(* CODESYS project LABELIX_849_HSC_Rtrig_24juillet.project
   CustomField04_name: CustomField04
   CustomField06_name: CustomField06
   CustomField07_name: CustomField07
   CustomField09_name: CustomField09
   CustomField08_name: CustomField08
   CustomField02_name: CustomField02
   CustomField05_name: CustomField05
   CustomField01_name: CustomField01
   CustomField03_name: CustomField03
   CustomField10_name: CustomField10

Project tree, tasks and I/O mapping:
  HMIS5T_REWIND : HMIS5T, Schneider Electric, order no. HMIS5T, version 2.0.3.24
    HMI Application
    COM1
      SoMachine_Network_Manager1 : SoMachine-Network_Manager, Schneider Electric, version 2.0.0.1
    USB
      SoMachine_Network_Manager3 : SoMachine-Network_Manager, Schneider Electric, version 2.0.0.1
    Ethernet
      SoMachine_Network_Manager2 : SoMachine-Network_Manager, Schneider Electric, version 2.0.0.1
  HMIS5T : HMIS5T, Schneider Electric, order no. HMIS5T, version 2.0.3.24
    HMI Application
    COM1
      SoMachine_Network_Manager4 : SoMachine-Network_Manager, Schneider Electric, version 2.0.0.1
    USB
      SoMachine_Network_Manager6 : SoMachine-Network_Manager, Schneider Electric, version 2.0.0.1
    Ethernet
      SoMachine_Network_Manager5 : SoMachine-Network_Manager, Schneider Electric, version 2.0.0.1
  MyController : TM258LF42DR, Schneider Electric, order no. TM258LF42DR, version 2.0.31.14
    application Application
      libraries: Toolbox, 2.0.3.1 (Schneider Electric)
      task MAST (cyclic, interval t#10ms, priority 2) calls PLC_PRG_LD_1
      task TaskMain (cyclic, interval t#20ms, priority 3) calls AccessCode, CAN_NETWORK, CONVERT, DRYER_1FD_3FX_STATIONS, ETH_NETWORK, FAULT_INTERLOCK, GRAVURE_PGM, LATCH_ERROR, Main, UNWIND_TENS_CTRL, COUNTER, UNWIND_TENS_CTRL, UW_FILT, UW_DIAM
      task Event_Task (externalevent, external event BLOCK0_I0, priority 1) calls EVENT_TASK
      COUNTER/
        program SPEED_DISPLAY [CFC]
        program PLC_PRG_LD_1 [LD]
        program speed_task [ST]
        program COUNTER [ST]
        program PLC_PRG_LD [LD]
      global variables GVL_OLD
      program Main [LD]
      global variables GVL_ARCHIVE
      global variables GVL_CAN_ARRAY
      program ETH_NETWORK [ST]
      global variables GVL_GENERAL
      program FAULT_INTERLOCK [LD]
      global variables GVL_ENCODER
      global variables GVL_NOT_USED_IOs
      global variables GVL_HMI
      program EVENT_TASK [ST]
      Symbols
      function HiddenPOU [ST]
      global variables GVL_ETHERNET
      data type stDryingGroup
      ErrorProvider
      program CONVERT [ST]
      program DRYER_1FD_3FX_STATIONS [LD]
      program CAN_NETWORK [ST]
      global variables GVL_KEEP_ARRAY
      program GRAVURE_PGM [LD]
      data type stTensionCtrlState
      global variables GVL_CONVERT
      data type stFlexoStation
      global variables GVL_KEY
      global variables GVL_DEBUG
      program LATCH_ERROR [LD]
      OPTIONS/
        program AccessCode [ST]
      UNWIND/
        program UW_FILT [LD]
        program UNWIND_TENS_CTRL [CFC]
        program UW_DIAM [ST]
      global variables GVL_counter
    Ethernet
        settings: IPAddress = [192, 168, 100, 202]; SubnetMask = [255, 255, 255, 0]; GatewayAddress = [192, 168, 100, 254]; WebServer = TRUE
      Modbus_TCP_Master : Modbus TCP Master, 3S - Smart Software Solutions GmbH, version 3.4.1.0
        GRAVURE : Modbus TCP Slave, 3S - Smart Software Solutions GmbH, version 3.4.0.0
            settings: IPAddress = [192, 168, 100, 208]; GravureWrite.Function Code = 16; GravureWrite.Read Offset = 0; GravureWrite.Read Length = 0; GravureWrite.Write Offset = 16#072C; GravureWrite.Write Length = 4; GravureWrite.Cycle Time = 100
            output wPar1837_GravureOn_ETH : WORD  // GravureWrite
            output wPar1838_GravureProcessOn_ETH : WORD  // GravureWrite
            output wPar1839_GravureFWD_ETH : WORD  // GravureWrite
            output wPar1840_GravureBCK_ETH : WORD  // GravureWrite
        REWIND_DF : Modbus TCP Slave, 3S - Smart Software Solutions GmbH, version 3.4.0.0
            settings: IPAddress = [192, 168, 100, 210]; REWIND_READ.Function Code = 3; REWIND_READ.Read Offset = 16#07E2; REWIND_READ.Read Length = 1; REWIND_READ.Write Offset = 0; REWIND_READ.Write Length = 0; REWIND_READ.Cycle Time = 100; RewindON.Function Code = 16; RewindON.Read Offset = 0; RewindON.Read Length = 0; RewindON.Write Offset = 16#072C; RewindON.Write Length = 2; RewindON.Cycle Time = 100; REWIND_STATE.Function Code = 3; REWIND_STATE.Read Offset = 16#03E8; REWIND_STATE.Read Length = 3; REWIND_STATE.Write Offset = 0; REWIND_STATE.Write Length = 0; REWIND_STATE.Cycle Time = 100
            input  wPar2019_DryPermit_ETH : WORD  // REWIND_READ
            output wPar1837_RewindOn_ETH : WORD  // RewindON
            output wPar1838_PidOn_ETH : WORD  // RewindON
            input  wPar1001_RewindHealthy_ETH : WORD  // REWIND_STATE
            input  wPar1002_RewindActive_ETH : WORD  // REWIND_STATE
            input  wPar1003_RewindZeroSpd_ETH : WORD  // REWIND_STATE
        REWIND : Modbus TCP Slave, 3S - Smart Software Solutions GmbH, version 3.4.0.0
            settings: IPAddress = [192, 168, 100, 204]; REWIND_READ.Function Code = 3; REWIND_READ.Read Offset = 16#07E2; REWIND_READ.Read Length = 1; REWIND_READ.Write Offset = 0; REWIND_READ.Write Length = 0; REWIND_READ.Cycle Time = 100; RewindON.Function Code = 16; RewindON.Read Offset = 0; RewindON.Read Length = 0; RewindON.Write Offset = 16#072C; RewindON.Write Length = 2; RewindON.Cycle Time = 100; REWIND_STATE.Function Code = 3; REWIND_STATE.Read Offset = 16#03E8; REWIND_STATE.Read Length = 3; REWIND_STATE.Write Offset = 0; REWIND_STATE.Write Length = 0; REWIND_STATE.Cycle Time = 100
            input  wPar2019_DryPermit_ETH : WORD  // REWIND_READ
            output wPar1837_RewindOn_ETH : WORD  // RewindON
            output wPar1838_PidOn_ETH : WORD  // RewindON
            input  wPar1001_RewindHealthy_ETH : WORD  // REWIND_STATE
            input  wPar1002_RewindActive_ETH : WORD  // REWIND_STATE
            input  wPar1003_RewindZeroSpd_ETH : WORD  // REWIND_STATE
        INFEED : Modbus TCP Slave, 3S - Smart Software Solutions GmbH, version 3.4.0.0
            settings: IPAddress = [192, 168, 100, 203]; Channel 2.Function Code = 16; Channel 2.Read Offset = 0; Channel 2.Read Length = 0; Channel 2.Write Offset = 16#072C; Channel 2.Write Length = 2; Channel 2.Cycle Time = 100; ALL_UnidriveSPs.Function Code = 3; ALL_UnidriveSPs.Read Offset = 16#07EF; ALL_UnidriveSPs.Read Length = 1; ALL_UnidriveSPs.Write Offset = 0; ALL_UnidriveSPs.Write Length = 0; ALL_UnidriveSPs.Cycle Time = 100; INFEED_STATE.Function Code = 3; INFEED_STATE.Read Offset = 16#03E8; INFEED_STATE.Read Length = 3; INFEED_STATE.Write Offset = 0; INFEED_STATE.Write Length = 0; INFEED_STATE.Cycle Time = 100; CounterReached_ETH.Function Code = 3; CounterReached_ETH.Read Offset = 16#078C; CounterReached_ETH.Read Length = 1; CounterReached_ETH.Write Offset = 0; CounterReached_ETH.Write Length = 0; CounterReached_ETH.Cycle Time = 100
            output wPar1837_InfeedOn_ETH : WORD  // Channel 2
            output wPar1838_FilterOn_ETH : WORD  // Channel 2
            input  wReadReg2031 : WORD  // ALL_UnidriveSPs
            input  wPar1001_InfeedHealthy_ETH : WORD  // INFEED_STATE
            input  wPar1002_InfeedActive_ETH : WORD  // INFEED_STATE
            input  wPar1003_InfeedZeroSpd_ETH : WORD  // INFEED_STATE
            input  wPar1933_CountReach_ETH : WORD  // CounterReached_ETH
        ANILOX_2 : Modbus TCP Slave, 3S - Smart Software Solutions GmbH, version 3.4.0.0
            settings: IPAddress = [192, 168, 100, 207]; AniloxWrite.Function Code = 16; AniloxWrite.Read Offset = 0; AniloxWrite.Read Length = 0; AniloxWrite.Write Offset = 16#072C; AniloxWrite.Write Length = 4; AniloxWrite.Cycle Time = 100
            output wPar1837_AniloxOn_2_ETH : WORD  // AniloxWrite
            output wPar1838_ProcessOn_2_ETH : WORD  // AniloxWrite
            output wPar1839_AniloxFWD_2_ETH : WORD  // AniloxWrite
            output wPar1840_AniloxBCK_2_ETH : WORD  // AniloxWrite
        TOP_REWIND : Modbus TCP Slave, 3S - Smart Software Solutions GmbH, version 3.4.0.0
            settings: IPAddress = [192, 168, 100, 205]; TOP_REWIND_READ.Function Code = 3; TOP_REWIND_READ.Read Offset = 16#07E2; TOP_REWIND_READ.Read Length = 1; TOP_REWIND_READ.Write Offset = 0; TOP_REWIND_READ.Write Length = 0; TOP_REWIND_READ.Cycle Time = 100; TopRewindON.Function Code = 16; TopRewindON.Read Offset = 0; TopRewindON.Read Length = 0; TopRewindON.Write Offset = 16#072C; TopRewindON.Write Length = 2; TopRewindON.Cycle Time = 100; TOP_REWIND_STATE.Function Code = 3; TOP_REWIND_STATE.Read Offset = 16#03E8; TOP_REWIND_STATE.Read Length = 3; TOP_REWIND_STATE.Write Offset = 0; TOP_REWIND_STATE.Write Length = 0; TOP_REWIND_STATE.Cycle Time = 100
            input  wPar2019 : WORD  // TOP_REWIND_READ
            output wPar1837_TopRewindOn_ETH : WORD  // TopRewindON
            output wPar1838_TopPidOn_ETH : WORD  // TopRewindON
            input  wPar1001_TopRewindHealthy_ETH : WORD  // TOP_REWIND_STATE
            input  wPar1002_TopRewindActive_ETH : WORD  // TOP_REWIND_STATE
            input  wPar1003_TopRewindZeroSpd_ETH : WORD  // TOP_REWIND_STATE
        REXROTH_1 : Modbus TCP Slave, 3S - Smart Software Solutions GmbH, version 3.4.0.0
            settings: IPAddress = [192, 168, 100, 211]; Channel 1.Function Code = 3; Channel 1.Read Offset = 16#0000; Channel 1.Read Length = 10; Channel 1.Write Offset = 0; Channel 1.Write Length = 0; Channel 1.Cycle Time = 100; Channel 2.Function Code = 16; Channel 2.Read Offset = 0; Channel 2.Read Length = 0; Channel 2.Write Offset = 16#000A; Channel 2.Write Length = 10; Channel 2.Cycle Time = 100
            output bGravureComTriggerRead : BIT  // Channel 1
            input  wInfeedManualGearing_ETH_i : WORD  // Channel 1
            input  wGravureGearingAdjust : WORD  // Channel 1
            input  bGravure_StatusDisabled_HMI_q2 : BOOL  // Channel 1.Bit 0
            input  bGravure_StatusSlowRot_HMI_q2 : BOOL  // Channel 1.Bit 1
            input  bGravure_StatusSynch_HMI_q2 : BOOL  // Channel 1.Bit 2
            input  bGravure_StatusError_HMI_q2 : BOOL  // Channel 1.Bit 3
            input  wDeviation_low_gb : WORD  // Channel 1
            input  wDeviation_high_gb : WORD  // Channel 1
            input  wRegiCtrlSetpoint_low_gb : WORD  // Channel 1
            input  wRegiCtrlSetpoint_high_gb : WORD  // Channel 1
            input  wLoadcellTension_low_gb : WORD  // Channel 1
            input  wLoadcellTension_high_gb : WORD  // Channel 1
            input  bInfeed_StatusDisabled_ETH_q : BOOL  // Channel 1.Bit 0
            input  bInfeed_StatusSlowRot_ETH_q : BOOL  // Channel 1.Bit 1
            input  bInfeed_StatusSynch_ETH_q : BOOL  // Channel 1.Bit 2
            input  bInfeed_StatusError_ETH_q : BOOL  // Channel 1.Bit 3
            output bGravureComTriggerWrite : BIT  // Channel 2
            output bGravure_Tens_Inc_ETH_q : BOOL  // Channel 2.Bit 0
            output bGravure_Tens_Dec_ETH_q : BOOL  // Channel 2.Bit 1
            output bGravure_Reg_Adv_ETH_q : BOOL  // Channel 2.Bit 2
            output bGravure_Reg_Ret_ETH_q : BOOL  // Channel 2.Bit 3
            output bGravureOn_ETH_q : BOOL  // Channel 2.Bit 4
            output bGravure_ResetDrive_HMI_q : BOOL  // Channel 2.Bit 5
            output bRewindPID_Out : BOOL  // Channel 2.Bit 6
            output bGravureSlowRot_ETH_q : BOOL  // Channel 2.Bit 7
            output bGravureRegiOn_HMI_q : BOOL  // Channel 2.Bit 8
            output bGravure_Jog_Adv_HMI_q : BOOL  // Channel 2.Bit 9
            output bGravure_Jog_Ret_HMI_q : BOOL  // Channel 2.Bit 10
            output bInfeedRegiOn_HMI_q : BOOL  // Channel 2.Bit 11
            output bInfeed_Tens_Inc_ETH_i : BOOL  // Channel 2.Bit 0
            output bInfeed_Tens_dec_ETH_i : BOOL  // Channel 2.Bit 1
            output bInfeedOn_ETH_i : BOOL  // Channel 2.Bit 2
            output bInfeed_Manual_ETH_i : BOOL  // Channel 2.Bit 3
            output bInfeed_ResetDrive_ETH_i : BOOL  // Channel 2.Bit 4
            output wRegAdjustStep_low_gb : WORD  // Channel 2
            output wRegAdjustStep_high_gb : WORD  // Channel 2
            unmapped channels: Channel 1, Channel 1, Channel 2, Channel 2, Channel 2, Channel 2, Channel 2, Channel 2, Channel 2, Channel 2
        ANILOX_1 : Modbus TCP Slave, 3S - Smart Software Solutions GmbH, version 3.4.0.0
            settings: IPAddress = [192, 168, 100, 206]; AniloxWrite.Function Code = 16; AniloxWrite.Read Offset = 0; AniloxWrite.Read Length = 0; AniloxWrite.Write Offset = 16#072C; AniloxWrite.Write Length = 4; AniloxWrite.Cycle Time = 100
            output wPar1837_AniloxOn_ETH : WORD  // AniloxWrite
            output wPar1838_ProcessOn_ETH : WORD  // AniloxWrite
            output wPar1839_AniloxFWD_ETH : WORD  // AniloxWrite
            output wPar1840_AniloxBCK_ETH : WORD  // AniloxWrite
    CAN0
      CANopen_Performance : CANopen Performance, Schneider Electric, order no. 1806, version 3.0.0.9
          settings: Enable Sync generation = FALSE; Enable Heartbeat generation = FALSE
        STATION_BOARD1 : OTB 1C0DM9LP, Schneider Electric, order no. 65275, version ProductVersion=0, ProductRevision=65537, Filename=SEOTB1C0DM9LP_0100E, FileVersion=1, FileRevision=0
            settings: General Options.Optional Device = TRUE; General Options.Not initialize = TRUE; NODEIDSAVED = 21; SDO Timeout = 1000000; EXPERTSETTINGS = True; Emergency-General Parameters.Emergency enabled = FALSE; Emergency-General Parameters.Emergency COBID = 16#95; Heartbeat-Producer Time = 200; PDO 16#1400.COBID = 16#00000215; PDO 16#1401.COBID = 16#80000315; PDO 16#1402.COBID = 16#80000415; PDO 16#1403.COBID = 16#80000515; PDO 16#1800.COBID = 16#00000195; PDO 16#1801.COBID = 16#80000295; PDO 16#1802.COBID = 16#80000395; PDO 16#1803.COBID = 16#80000495; Word Write Output 0 to 7.Index = 16#6300; Word Write Output 0 to 7.Subindex = 16#01; Word Write Output 0 to 7.ObjectLength = 16; Word Read Input 0 to 11.Index = 16#6100; Word Read Input 0 to 11.Subindex = 16#01; Word Read Input 0 to 11.ObjectLength = 16; Number of SDO = 33; Set Guardtime.Index = 16#100C; Set Guardtime.Subindex = 16#00; Set Guardtime.Value = 16#00000000; Set Guardtime.Size = 16; Set Guardtime.AbortIfError = FALSE; Set Guardtime.JumpToLine = FALSE; Set Guardtime.Line = 0; Set Lifetime.Index = 16#100D; Set Lifetime.Subindex = 16#00; Set Lifetime.Value = 16#00000000; Set Lifetime.Size = 8; Set Lifetime.AbortIfError = FALSE; Set Lifetime.JumpToLine = FALSE; Set Lifetime.Line = 0; Set Emcy CobID.Index = 16#1014; Set Emcy CobID.Subindex = 16#00; Set Emcy CobID.Value = 16#80000095;
              Set Emcy CobID.Size = 32; Set Emcy CobID.AbortIfError = FALSE; Set Emcy CobID.JumpToLine = FALSE; Set Emcy CobID.Line = 0; Set Heartbeat Consumer.Index = 16#1016; Set Heartbeat Consumer.Subindex = 16#01; Set Heartbeat Consumer.Value = 0; Set Heartbeat Consumer.Size = 32; Set Heartbeat Consumer.AbortIfError = FALSE; Set Heartbeat Consumer.JumpToLine = FALSE; Set Heartbeat Consumer.Line = 0; Set Heartbeat Producer.Index = 16#1017; Set Heartbeat Producer.Subindex = 16#00; Set Heartbeat Producer.Value = 16#000000C8; Set Heartbeat Producer.Size = 16; Set Heartbeat Producer.AbortIfError = FALSE; Set Heartbeat Producer.JumpToLine = FALSE; Set Heartbeat Producer.Line = 0; Disable PDO.Index = 16#1400; Disable PDO.Subindex = 16#01; Disable PDO.Value = 16#80000215; Disable PDO.Size = 32; Disable PDO.AbortIfError = FALSE; Disable PDO.JumpToLine = FALSE; Disable PDO.Line = 0; Set transmission type.Index = 16#1400; Set transmission type.Subindex = 16#02; Set transmission type.Value = 16#FF; Set transmission type.Size = 8; Set transmission type.AbortIfError = FALSE; Set transmission type.JumpToLine = FALSE; Set transmission type.Line = 0; Clear pdo mapping.Index = 16#1600; Clear pdo mapping.Subindex = 16#00; Clear pdo mapping.Value = 16#0; Clear pdo mapping.Size = 8; Clear pdo mapping.AbortIfError = FALSE; Clear pdo mapping.JumpToLine = FALSE; Clear pdo mapping.Line = 0; Set Mapping.Index = 16#1600;
              Set Mapping.Subindex = 16#01; Set Mapping.Value = 16#63000110; Set Mapping.Size = 32; Set Mapping.AbortIfError = FALSE; Set Mapping.JumpToLine = FALSE; Set Mapping.Line = 0; Set number of pdos.Index = 16#1600; Set number of pdos.Subindex = 16#00; Set number of pdos.Value = 16#01; Set number of pdos.Size = 8; Set number of pdos.AbortIfError = FALSE; Set number of pdos.JumpToLine = FALSE; Set number of pdos.Line = 0; Set and enable COB-ID.Index = 16#1400; Set and enable COB-ID.Subindex = 16#01; Set and enable COB-ID.Value = 16#00000215; Set and enable COB-ID.Size = 32; Set and enable COB-ID.AbortIfError = FALSE; Set and enable COB-ID.JumpToLine = FALSE; Set and enable COB-ID.Line = 0; Disable PDO.Index = 16#1401; Disable PDO.Subindex = 16#01; Disable PDO.Value = 16#80000315; Disable PDO.Size = 32; Disable PDO.AbortIfError = FALSE; Disable PDO.JumpToLine = FALSE; Disable PDO.Line = 0; Disable PDO.Index = 16#1402; Disable PDO.Subindex = 16#01; Disable PDO.Value = 16#80000415; Disable PDO.Size = 32; Disable PDO.AbortIfError = FALSE; Disable PDO.JumpToLine = FALSE; Disable PDO.Line = 0; Disable PDO.Index = 16#1403; Disable PDO.Subindex = 16#01; Disable PDO.Value = 16#80000515; Disable PDO.Size = 32; Disable PDO.AbortIfError = FALSE; Disable PDO.JumpToLine = FALSE;
              Disable PDO.Line = 0; Disable PDO.Index = 16#1404; Disable PDO.Subindex = 16#01; Disable PDO.Value = 16#80000001; Disable PDO.Size = 32; Disable PDO.AbortIfError = FALSE; Disable PDO.JumpToLine = FALSE; Disable PDO.Line = 0; Disable PDO.Index = 16#1405; Disable PDO.Subindex = 16#01; Disable PDO.Value = 16#80000001; Disable PDO.Size = 32; Disable PDO.AbortIfError = FALSE; Disable PDO.JumpToLine = FALSE; Disable PDO.Line = 0; Disable PDO.Index = 16#1406; Disable PDO.Subindex = 16#01; Disable PDO.Value = 16#80000001; Disable PDO.Size = 32; Disable PDO.AbortIfError = FALSE; Disable PDO.JumpToLine = FALSE; Disable PDO.Line = 0; Disable PDO.Index = 16#1407; Disable PDO.Subindex = 16#01; Disable PDO.Value = 16#80000001; Disable PDO.Size = 32; Disable PDO.AbortIfError = FALSE; Disable PDO.JumpToLine = FALSE; Disable PDO.Line = 0; Disable PDO.Index = 16#1800; Disable PDO.Subindex = 16#01; Disable PDO.Value = 16#80000195; Disable PDO.Size = 32; Disable PDO.AbortIfError = FALSE; Disable PDO.JumpToLine = FALSE; Disable PDO.Line = 0; Set transmission type.Index = 16#1800; Set transmission type.Subindex = 16#02; Set transmission type.Value = 16#FF; Set transmission type.Size = 8;
              Set transmission type.AbortIfError = FALSE; Set transmission type.JumpToLine = FALSE; Set transmission type.Line = 0; Set inhibit time.Index = 16#1800; Set inhibit time.Subindex = 16#03; Set inhibit time.Value = 16#0000; Set inhibit time.Size = 16; Set inhibit time.AbortIfError = FALSE; Set inhibit time.JumpToLine = FALSE; Set inhibit time.Line = 0; Set event time.Index = 16#1800; Set event time.Subindex = 16#05; Set event time.Value = 16#0000; Set event time.Size = 16; Set event time.AbortIfError = FALSE; Set event time.JumpToLine = FALSE; Set event time.Line = 0; Clear pdo mapping.Index = 16#1A00; Clear pdo mapping.Subindex = 16#00; Clear pdo mapping.Value = 16#0; Clear pdo mapping.Size = 8; Clear pdo mapping.AbortIfError = FALSE; Clear pdo mapping.JumpToLine = FALSE; Clear pdo mapping.Line = 0; Set Mapping.Index = 16#1A00; Set Mapping.Subindex = 16#01; Set Mapping.Value = 16#61000110; Set Mapping.Size = 32; Set Mapping.AbortIfError = FALSE; Set Mapping.JumpToLine = FALSE; Set Mapping.Line = 0; Set number of pdos.Index = 16#1A00; Set number of pdos.Subindex = 16#00; Set number of pdos.Value = 16#01; Set number of pdos.Size = 8; Set number of pdos.AbortIfError = FALSE; Set number of pdos.JumpToLine = FALSE; Set number of pdos.Line = 0; Set and enable COB-ID.Index = 16#1800; Set and enable COB-ID.Subindex = 16#01;
              Set and enable COB-ID.Value = 16#00000195; Set and enable COB-ID.Size = 32; Set and enable COB-ID.AbortIfError = FALSE; Set and enable COB-ID.JumpToLine = FALSE; Set and enable COB-ID.Line = 0; Disable PDO.Index = 16#1801; Disable PDO.Subindex = 16#01; Disable PDO.Value = 16#80000295; Disable PDO.Size = 32; Disable PDO.AbortIfError = FALSE; Disable PDO.JumpToLine = FALSE; Disable PDO.Line = 0; Disable PDO.Index = 16#1802; Disable PDO.Subindex = 16#01; Disable PDO.Value = 16#80000395; Disable PDO.Size = 32; Disable PDO.AbortIfError = FALSE; Disable PDO.JumpToLine = FALSE; Disable PDO.Line = 0; Disable PDO.Index = 16#1803; Disable PDO.Subindex = 16#01; Disable PDO.Value = 16#80000495; Disable PDO.Size = 32; Disable PDO.AbortIfError = FALSE; Disable PDO.JumpToLine = FALSE; Disable PDO.Line = 0; Disable PDO.Index = 16#1804; Disable PDO.Subindex = 16#01; Disable PDO.Value = 16#80000001; Disable PDO.Size = 32; Disable PDO.AbortIfError = FALSE; Disable PDO.JumpToLine = FALSE; Disable PDO.Line = 0; Disable PDO.Index = 16#1805; Disable PDO.Subindex = 16#01; Disable PDO.Value = 16#80000001; Disable PDO.Size = 32; Disable PDO.AbortIfError = FALSE; Disable PDO.JumpToLine = FALSE; Disable PDO.Line = 0;
              Disable PDO.Index = 16#1806; Disable PDO.Subindex = 16#01; Disable PDO.Value = 16#80000001; Disable PDO.Size = 32; Disable PDO.AbortIfError = FALSE; Disable PDO.JumpToLine = FALSE; Disable PDO.Line = 0; Disable PDO.Index = 16#1807; Disable PDO.Subindex = 16#01; Disable PDO.Value = 16#80000001; Disable PDO.Size = 32; Disable PDO.AbortIfError = FALSE; Disable PDO.JumpToLine = FALSE; Disable PDO.Line = 0
            output Application.GVL_CAN_ARRAY.wStationBrd_LED_q[1] : UINT  // Word Write Output 0 to 7
            input  Application.GVL_CAN_ARRAY.wArStationBrd[1] : UINT  // Word Read Input 0 to 11
        STATION_BOARD2 : OTB 1C0DM9LP, Schneider Electric, order no. 65275, version ProductVersion=0, ProductRevision=65537, Filename=SEOTB1C0DM9LP_0100E, FileVersion=1, FileRevision=0
            settings: General Options.Optional Device = TRUE; General Options.Not initialize = TRUE; NODEIDSAVED = 22; SDO Timeout = 1000000; EXPERTSETTINGS = True; Sync-General Parameters.Sync-COBID = 16#00000080; Sync-General Parameters.Communication Cycle Period = 16#0000C350 usec; Emergency-General Parameters.Emergency enabled = FALSE; Emergency-General Parameters.Emergency COBID = 16#96; Heartbeat-Producer Time = 200; PDO 16#1400.COBID = 16#00000216; PDO 16#1401.COBID = 16#80000182; Generic COBID = '16#80000182'; PDO 16#1402.COBID = 16#80000416; PDO 16#1403.COBID = 16#80000516; PDO 16#1800.COBID = 16#00000196; PDO 16#1801.COBID = 16#80000182; Generic COBID = '16#80000182'; PDO 16#1802.COBID = 16#80000396; PDO 16#1803.COBID = 16#80000496; Word Write Output 16 to 31.Index = 16#6300; Word Write Output 16 to 31.Subindex = 16#02; Word Write Output 16 to 31.ObjectLength = 16; Word Read Input 16 to 31.Index = 16#6100; Word Read Input 16 to 31.Subindex = 16#02; Word Read Input 16 to 31.ObjectLength = 16; Number of SDO = 33; Set Guardtime.Index = 16#100C; Set Guardtime.Subindex = 16#00; Set Guardtime.Value = 16#00000000; Set Guardtime.Size = 16; Set Guardtime.AbortIfError = FALSE; Set Guardtime.JumpToLine = FALSE; Set Guardtime.Line = 0; Set Lifetime.Index = 16#100D; Set Lifetime.Subindex = 16#00; Set Lifetime.Value = 16#00000000; Set Lifetime.Size = 8; Set Lifetime.AbortIfError = FALSE; Set Lifetime.JumpToLine = FALSE;
              Set Lifetime.Line = 0; Set Emcy CobID.Index = 16#1014; Set Emcy CobID.Subindex = 16#00; Set Emcy CobID.Value = 16#80000096; Set Emcy CobID.Size = 32; Set Emcy CobID.AbortIfError = FALSE; Set Emcy CobID.JumpToLine = FALSE; Set Emcy CobID.Line = 0; Set Heartbeat Consumer.Index = 16#1016; Set Heartbeat Consumer.Subindex = 16#01; Set Heartbeat Consumer.Value = 0; Set Heartbeat Consumer.Size = 32; Set Heartbeat Consumer.AbortIfError = FALSE; Set Heartbeat Consumer.JumpToLine = FALSE; Set Heartbeat Consumer.Line = 0; Set Heartbeat Producer.Index = 16#1017; Set Heartbeat Producer.Subindex = 16#00; Set Heartbeat Producer.Value = 16#000000C8; Set Heartbeat Producer.Size = 16; Set Heartbeat Producer.AbortIfError = FALSE; Set Heartbeat Producer.JumpToLine = FALSE; Set Heartbeat Producer.Line = 0; Disable PDO.Index = 16#1400; Disable PDO.Subindex = 16#01; Disable PDO.Value = 16#80000216; Disable PDO.Size = 32; Disable PDO.AbortIfError = FALSE; Disable PDO.JumpToLine = FALSE; Disable PDO.Line = 0; Set transmission type.Index = 16#1400; Set transmission type.Subindex = 16#02; Set transmission type.Value = 16#FF; Set transmission type.Size = 8; Set transmission type.AbortIfError = FALSE; Set transmission type.JumpToLine = FALSE; Set transmission type.Line = 0; Clear pdo mapping.Index = 16#1600; Clear pdo mapping.Subindex = 16#00; Clear pdo mapping.Value = 16#0; Clear pdo mapping.Size = 8;
              Clear pdo mapping.AbortIfError = FALSE; Clear pdo mapping.JumpToLine = FALSE; Clear pdo mapping.Line = 0; Set Mapping.Index = 16#1600; Set Mapping.Subindex = 16#01; Set Mapping.Value = 16#63000210; Set Mapping.Size = 32; Set Mapping.AbortIfError = FALSE; Set Mapping.JumpToLine = FALSE; Set Mapping.Line = 0; Set number of pdos.Index = 16#1600; Set number of pdos.Subindex = 16#00; Set number of pdos.Value = 16#01; Set number of pdos.Size = 8; Set number of pdos.AbortIfError = FALSE; Set number of pdos.JumpToLine = FALSE; Set number of pdos.Line = 0; Set and enable COB-ID.Index = 16#1400; Set and enable COB-ID.Subindex = 16#01; Set and enable COB-ID.Value = 16#00000216; Set and enable COB-ID.Size = 32; Set and enable COB-ID.AbortIfError = FALSE; Set and enable COB-ID.JumpToLine = FALSE; Set and enable COB-ID.Line = 0; Disable PDO.Index = 16#1401; Disable PDO.Subindex = 16#01; Disable PDO.Value = 16#80000182; Disable PDO.Size = 32; Disable PDO.AbortIfError = FALSE; Disable PDO.JumpToLine = FALSE; Disable PDO.Line = 0; Disable PDO.Index = 16#1402; Disable PDO.Subindex = 16#01; Disable PDO.Value = 16#80000416; Disable PDO.Size = 32; Disable PDO.AbortIfError = FALSE; Disable PDO.JumpToLine = FALSE; Disable PDO.Line = 0; Disable PDO.Index = 16#1403; Disable PDO.Subindex = 16#01;
              Disable PDO.Value = 16#80000516; Disable PDO.Size = 32; Disable PDO.AbortIfError = FALSE; Disable PDO.JumpToLine = FALSE; Disable PDO.Line = 0; Disable PDO.Index = 16#1404; Disable PDO.Subindex = 16#01; Disable PDO.Value = 16#80000001; Disable PDO.Size = 32; Disable PDO.AbortIfError = FALSE; Disable PDO.JumpToLine = FALSE; Disable PDO.Line = 0; Disable PDO.Index = 16#1405; Disable PDO.Subindex = 16#01; Disable PDO.Value = 16#80000001; Disable PDO.Size = 32; Disable PDO.AbortIfError = FALSE; Disable PDO.JumpToLine = FALSE; Disable PDO.Line = 0; Disable PDO.Index = 16#1406; Disable PDO.Subindex = 16#01; Disable PDO.Value = 16#80000001; Disable PDO.Size = 32; Disable PDO.AbortIfError = FALSE; Disable PDO.JumpToLine = FALSE; Disable PDO.Line = 0; Disable PDO.Index = 16#1407; Disable PDO.Subindex = 16#01; Disable PDO.Value = 16#80000001; Disable PDO.Size = 32; Disable PDO.AbortIfError = FALSE; Disable PDO.JumpToLine = FALSE; Disable PDO.Line = 0; Disable PDO.Index = 16#1800; Disable PDO.Subindex = 16#01; Disable PDO.Value = 16#80000196; Disable PDO.Size = 32; Disable PDO.AbortIfError = FALSE; Disable PDO.JumpToLine = FALSE; Disable PDO.Line = 0;
              Set transmission type.Index = 16#1800; Set transmission type.Subindex = 16#02; Set transmission type.Value = 16#FF; Set transmission type.Size = 8; Set transmission type.AbortIfError = FALSE; Set transmission type.JumpToLine = FALSE; Set transmission type.Line = 0; Set inhibit time.Index = 16#1800; Set inhibit time.Subindex = 16#03; Set inhibit time.Value = 16#0000; Set inhibit time.Size = 16; Set inhibit time.AbortIfError = FALSE; Set inhibit time.JumpToLine = FALSE; Set inhibit time.Line = 0; Set event time.Index = 16#1800; Set event time.Subindex = 16#05; Set event time.Value = 16#0000; Set event time.Size = 16; Set event time.AbortIfError = FALSE; Set event time.JumpToLine = FALSE; Set event time.Line = 0; Clear pdo mapping.Index = 16#1A00; Clear pdo mapping.Subindex = 16#00; Clear pdo mapping.Value = 16#0; Clear pdo mapping.Size = 8; Clear pdo mapping.AbortIfError = FALSE; Clear pdo mapping.JumpToLine = FALSE; Clear pdo mapping.Line = 0; Set Mapping.Index = 16#1A00; Set Mapping.Subindex = 16#01; Set Mapping.Value = 16#61000210; Set Mapping.Size = 32; Set Mapping.AbortIfError = FALSE; Set Mapping.JumpToLine = FALSE; Set Mapping.Line = 0; Set number of pdos.Index = 16#1A00; Set number of pdos.Subindex = 16#00; Set number of pdos.Value = 16#01; Set number of pdos.Size = 8; Set number of pdos.AbortIfError = FALSE;
              Set number of pdos.JumpToLine = FALSE; Set number of pdos.Line = 0; Set and enable COB-ID.Index = 16#1800; Set and enable COB-ID.Subindex = 16#01; Set and enable COB-ID.Value = 16#00000196; Set and enable COB-ID.Size = 32; Set and enable COB-ID.AbortIfError = FALSE; Set and enable COB-ID.JumpToLine = FALSE; Set and enable COB-ID.Line = 0; Disable PDO.Index = 16#1801; Disable PDO.Subindex = 16#01; Disable PDO.Value = 16#80000182; Disable PDO.Size = 32; Disable PDO.AbortIfError = FALSE; Disable PDO.JumpToLine = FALSE; Disable PDO.Line = 0; Disable PDO.Index = 16#1802; Disable PDO.Subindex = 16#01; Disable PDO.Value = 16#80000396; Disable PDO.Size = 32; Disable PDO.AbortIfError = FALSE; Disable PDO.JumpToLine = FALSE; Disable PDO.Line = 0; Disable PDO.Index = 16#1803; Disable PDO.Subindex = 16#01; Disable PDO.Value = 16#80000496; Disable PDO.Size = 32; Disable PDO.AbortIfError = FALSE; Disable PDO.JumpToLine = FALSE; Disable PDO.Line = 0; Disable PDO.Index = 16#1804; Disable PDO.Subindex = 16#01; Disable PDO.Value = 16#80000001; Disable PDO.Size = 32; Disable PDO.AbortIfError = FALSE; Disable PDO.JumpToLine = FALSE; Disable PDO.Line = 0; Disable PDO.Index = 16#1805; Disable PDO.Subindex = 16#01; Disable PDO.Value = 16#80000001;
              Disable PDO.Size = 32; Disable PDO.AbortIfError = FALSE; Disable PDO.JumpToLine = FALSE; Disable PDO.Line = 0; Disable PDO.Index = 16#1806; Disable PDO.Subindex = 16#01; Disable PDO.Value = 16#80000001; Disable PDO.Size = 32; Disable PDO.AbortIfError = FALSE; Disable PDO.JumpToLine = FALSE; Disable PDO.Line = 0; Disable PDO.Index = 16#1807; Disable PDO.Subindex = 16#01; Disable PDO.Value = 16#80000001; Disable PDO.Size = 32; Disable PDO.AbortIfError = FALSE; Disable PDO.JumpToLine = FALSE; Disable PDO.Line = 0
            output Application.GVL_CAN_ARRAY.wStationBrd_LED_q[2] : UINT  // Word Write Output 16 to 31
            input  Application.GVL_CAN_ARRAY.wArStationBrd[2] : UINT  // Word Read Input 16 to 31
    PCI Slots
      <Empty>
      <Empty>
    Serial Line
      SoMachine_Network_Manager : SoMachine-Network_Manager, Schneider Electric, version 2.0.1.10
    TM5
      TM5_Manager : TM5 Manager, Schneider Electric, order no. TM5, version 2.0.2.3
        TM5SAO2L : TM5SAO2L, Schneider Electric, order no. TM5SAO2L, version 3.1.1.2
            output uiPID_Output_q : INT  // AnalogOutput00
            unmapped channels: AnalogOutput01
        TM5SAI2L : TM5SAI2L, Schneider Electric, order no. TM5SAI2L, version 3.1.1.2
            input  uiUNWIND_ACTUAL_TENSION : INT  // AnalogInput00
            unmapped channels: AnalogInput01, StatusInput00
        Embedded Bus
          DO6RE : DO6RE, Schneider Electric, order no. DO6RE, version 3.1.1.1
              output bHeater1A_q : BOOL  // DigitalOutputs.DigitalOutput00
              output bHeater1B_q : BOOL  // DigitalOutputs.DigitalOutput01
              output bHeater2A_q : BOOL  // DigitalOutputs.DigitalOutput02
              output bHeater2B_q : BOOL  // DigitalOutputs.DigitalOutput03
              output bEXH_q : BOOL  // DigitalOutputs.DigitalOutput04
              output bOscillateBlade_q : BOOL  // DigitalOutputs.DigitalOutput05
              unmapped channels: DigitalOutputs
          DO6RE_1 : DO6RE, Schneider Electric, order no. DO6RE, version 3.1.1.1
              output bRun_q : BOOL  // DigitalOutputs.DigitalOutput00
              output bJog_q : BOOL  // DigitalOutputs.DigitalOutput01
              output Application.ArFlexoStation[1].bRegAdvance_q : BOOL  // DigitalOutputs.DigitalOutput02
              output Application.ArFlexoStation[1].bRegRetard_q : BOOL  // DigitalOutputs.DigitalOutput03
              output Application.LATCH_ERROR.b_Gravure_q : BOOL  // DigitalOutputs.DigitalOutput04
              output bResetSpeed_q : BOOL  // DigitalOutputs.DigitalOutput05
              unmapped channels: DigitalOutputs
          DI6DE : DI6DE, Schneider Electric, order no. DI6DE, version 3.1.1.1
              input  bEmergency_i : BOOL  // DigitalInputs.DigitalInput00
              input  bRun_i : BOOL  // DigitalInputs.DigitalInput01
              input  bStop_i : BOOL  // DigitalInputs.DigitalInput02
              input  bJog_i : BOOL  // DigitalInputs.DigitalInput03
              input  Ovl_Exh_i : BOOL  // DigitalInputs.DigitalInput04
              input  Unwind_Coupling1_i : BOOL  // DigitalInputs.DigitalInput05
              unmapped channels: DigitalInputs
          D000E : D000E, Schneider Electric, order no. D000E, version 3.1.1.1
          DI6DE_1 : DI6DE, Schneider Electric, order no. DI6DE, version 3.1.1.1
              input  Application.LATCH_ERROR.b_Gravure_i : BOOL  // DigitalInputs.DigitalInput01
              input  bAllDrivesHealthy_i : BOOL  // DigitalInputs.DigitalInput04
              input  bMainDriveHealthy_i : BOOL  // DigitalInputs.DigitalInput05
              unmapped channels: DigitalInputs
        TM5SDO4R : TM5SDO4R, Schneider Electric, order no. TM5SDO4R, version 3.1.1.1
            output bGravureKickoff_q : BOOL  // DigitalOutputs.DigitalOutput00
            unmapped channels: DigitalOutputs
    Expert
      DM72F1 : DM72F1, Schneider Electric, order no. DM72F1, version 2.0.31.14
          settings: Synchronization.Output process task = 'MAST'
          output bIncSpeed_q : BOOL  // QB0.Q0
          output bDecSpeed_q : BOOL  // QB0.Q1
          unmapped channels: IB0, IB1, QB0
        HSCMain1 : HSCMain, Schneider Electric, order no. HSCMain, version 2.0.31.14
      PowerDistribution : POWER, Schneider Electric, order no. POWER, version 2.0.31.14
          unmapped channels: IB0
      DM72F0 : DM72F0, Schneider Electric, order no. DM72F0, version 2.0.31.14
          settings: Synchronization.Output process task = 'MAST'
          input  bEndOfRoll_i : BOOL  // IB0.I0
          input  bLineShaft_i : BOOL  // IB0.I1
          input  bThermo1_i : BOOL  // IB0.I2
          input  bThermo2_i : BOOL  // IB0.I3
          input  bMinSpeed_i : BOOL  // IB0.I5
          input  bZeroSpeed_i : BOOL  // IB0.I6
          output bBuzzer_q : BOOL  // QB0.Q0
          output bWebGripper_q : BOOL  // QB0.Q1
          unmapped channels: IB0, IB1, QB0
        Event_Latch0 : Event_Latch0, Schneider Electric, order no. EventLatch0, version 2.0.31.14
  MachineLayoutPicture
*)

// MyController/Application/stDryingGroup
TYPE stDryingGroup :
STRUCT

	bDryOff_i:BOOL;
	bBlowerOn_i:BOOL;
	bLowHeatOn_i:BOOL;
	bHighHeatOn_i:BOOL;

	bHeaterA_q:BOOL;	//FIRST HEATING ELEMENT
	bHeaterB_q:BOOL;	//SECOND HEATING ELEMENT
	
	bFD_q:BOOL;			//Forced Draft Dryer
END_STRUCT
END_TYPE

// MyController/Application/stTensionCtrlState
TYPE stTensionCtrlState :
STRUCT
	
	bOffMode:BOOL:=0;
	bManualMode:BOOL:=1;
	bAutoMode:BOOL:=0;
END_STRUCT
END_TYPE

// MyController/Application/stFlexoStation
TYPE stFlexoStation :
STRUCT

				//INPUTS
				bAniloxMtr		:BOOL;
				bAniloxKickOff	:BOOL;
				
				bPlateKickoff	:BOOL;
				bInfraRed		:BOOL;
				bRegAdvance		:BOOL;
				bRegRetard		:BOOL;
				bRunPlus		:BOOL;
				bRunMinus		:BOOL;
				bJog			:BOOL;
				bStop			:BOOL;
				bSetup			:BOOL;
				bInkingOn		:BOOL;
				bPrintingOn 	:BOOL;
				
				bSpare1			:BOOL;
				bSpare2			:BOOL;
				bSpare3			:BOOL;
				//OUTPUTS
				bRegAdvance_q		:BOOL;
				bRegRetard_q		:BOOL;
				bAniloxMot_q		:BOOL;
				bPlateKickoff_q		:BOOL;
				bAniloxKickoff_q	:BOOL;
				
				bSpare1_q			:BOOL;
				bSpare2_q			:BOOL;
				bSpare3_q			:BOOL;
				
END_STRUCT
END_TYPE

// MyController/Application/GVL_OLD
VAR_GLOBAL

//uiStationBrd1_gb:UINT;
//bAniloxMotor1_gb:BOOL;


//uiStationBrd2_gb:UINT;
//uiStationBrd3_gb:UINT;
//uiStationBrd4_gb:UINT;

wStationBrd1_gb:WORD;
wStationBrd2_gb:WORD;
wStationBrd3_gb:WORD;
wStationBrd4_gb:WORD;
wStationBrd5_gb:WORD;
wStationBrd6_gb:WORD;
wStationBrd7_gb:WORD;
wStationBrd8_gb:WORD;
wStationBrd9_gb:WORD;
wStationBrd10_gb:WORD;



wStationBrd1_LED_q:WORD;
wStationBrd2_LED_q:WORD;
wStationBrd3_LED_q:WORD;
wStationBrd4_LED_q:WORD;
wStationBrd5_LED_q:WORD;
wStationBrd6_LED_q:WORD;
wStationBrd7_LED_q:WORD;
wStationBrd8_LED_q:WORD;
wStationBrd9_LED_q:WORD;
wStationBrd10_LED_q:WORD;

END_VAR

// MyController/Application/GVL_ARCHIVE
VAR_GLOBAL


	bSafetyGuard_i:		BOOL	:=	TRUE;
	//bUnwindCoupling_i:	BOOL	:=	TRUE;
	//bUnwindLiftArm_i:	BOOL	:=	TRUE;
	bRewindCoupling_i:	BOOL	:=	TRUE;
	//bRewindLiftArm_i:		BOOL	:=	TRUE;

	
	//bAniloxMot1_q:		BOOL;
	//bAniloxMot2_q:		BOOL;
	bAniloxMot1_1_q		:BOOL;
	bAniloxMot1_2_q		:BOOL;
	
	
	bWebClean_i			:BOOL;
	bWebCleanStick_q	:BOOL;
	bWebCleanNip_q		:BOOL;
	bHeaterThermal_i	:BOOL;
	
	
	
	bEXH_Healthy_i		:BOOL;
	Ovl_Fd_i:BOOL;
	
	//bIncSpeed_q:BOOL;
	//bDecSpeed_q:BOOL;
END_VAR

// MyController/Application/GVL_CAN_ARRAY
VAR_GLOBAL

	
	
	wArStationBrd: ARRAY[1..20]OF WORD;
	
	wStationBrd_LED_q: ARRAY[1..20]OF WORD;
	
	ArFlexoStation: ARRAY[1..20]OF stFlexoStation;
	



	
	wRelayBrd_OUT_q: ARRAY[1..20]OF WORD;
	wRelayBrd_IN_q: ARRAY[1..20]OF WORD;
	//OUTPUT ARRAYS
	
	
	
	bGreenLightRunStatus_q:BOOL;
	
END_VAR

// MyController/Application/GVL_GENERAL
VAR_GLOBAL

	//bMinSpeed_i: BOOL;
	
	okToJog: BOOL;
    intRun: BOOL;
	intJog: BOOL;
	jogTimeLimit: BOOL;
	RunTimeLimit: BOOL;
	timerBuzzer: TON;
	Timer1: TOF;
	rewindTimerOffdel: TON;
	//mainDriveOndel: TON;
	rejogTimer: TON;
	zeroSpeedOndel: TON;			
	pid1: PID;
    driveSignal: INT;
	timerPlate:Ton;
	heatEnable: BOOL;
	
	timerFD1: TON;
	timerFD2: TON;
	timerFD3: TON;
	timerFD4: TON;
	timerFD5: TON;
	
	uvBlowerOvlLtch: BOOL;
	resetFaultTS: BOOL;
	uvLampOverhLtch: BOOL;
	uvLampOutLtch: BOOL;
	uvOvercurrentLtch: BOOL;
	uvPsOvertempLtch: BOOL;
	emerTS: BOOL;
	emerComb: BOOL;
	uvOkToGo: BOOL;
	uvOnTS: BOOL;
	shutterTestTS: BOOL;
	shutterTestLtch: BOOL;
	TimerShutterTest: TON;
	timerUVBlowerOffdel: TON;
    timerUVBlowerOnDel: TON;
    shutterOk: BOOL;
	shutterOkLtch: BOOL;
	TimerShutterOk: TON;
	shutterFaultLtch: BOOL;
	uvAnalogSignalMin: BOOL;
	uvAnalogSignalVar: BOOL;
		tempProbeReal: REAL;
	FreqMeasure1: FREQ_MEASURE;
	frequencyReal: REAL;

		SR_AniloxSv: SR;
	SR_Infeed: SR;
	setupActive: BOOL;
	SR_RewindOn: SR;
	SR_TopRewindOn: SR;
	SR_GravureOn: SR;
	//bGravureComTrigger: BOOL;


	COUNTER_REACHED:BOOL;
	
	SR_RewindStart: SR;
	SR_JogTimeLimit: SR;
	SR_SetupActive: SR;
	SR_EndRollInd: SR;
	
    SR_FD1: SR;
	SR_FD2: SR;
	SR_FD3: SR;
	SR_FD4: SR;
	SR_FD5: SR;
	
	SR_EXH: SR;
	
	
	SR_InkinkOn: SR;
	SR_PrintingOn: SR;
	SR_PlateSVOut: SR;
		SR_uvBlowerOvl: SR;
	SR_uvLampOverheat: SR;
	SR_uvLampOut: SR;
		SR_uvOvercurrent: SR;
	SR_uvPsOvertemp: SR;
	SR_ShutterOk: SR;
	SR_ShutterFault: SR;
	SR_uvLampOn: SR;
	SR_uvBlower: SR;
	SR_uvShutterTest: SR;
	uvSetpointReal: REAL;
	uvSetpointReal100: REAL;
	uvSetpointInt100: INT;
	driveSignalReal: REAL;
		
	uvBlowerTimeLeft: TIME;
	blink2: BLINK;
	shutterMonitor: BOOL;
		
	TransitOnToWarmup: TON;
	TransitWarmupToReady: TON;
	noMinSpeedBuffer: TON;
	SR_WarmupFail: SR;
	warmupFailLatch: BOOL;
	SR_ReadyFailLatch: SR;
	readyFailLatch: BOOL;
	timeOutDisplay: BOOL;
	timeOut: BOOL;
	uvWarmupDisplay: BOOL;
	SR_uvACVoltagePresent: SR;
	uvACVoltageFaultLatch: BOOL;
	tempsetpointFReal: REAL;
	tempSetpointCReal: REAL;
		tempProbeCx10Real: REAL;
	tempDisplayFReal: REAL;
	tempSetpointCx10Real: REAL;
	//bAniloxMotor_1: BOOL;
	
	bRun_gb:BOOL;
	bJog_gb:BOOL;
	bStop_gb:BOOL;
	
	
	

	
	bInkingOn_gb: BOOL := FALSE;
	bPrintingOn_gb: BOOL := FALSE;
	bSetup_gb: BOOL := FALSE;
	
	
	
	heaterOnOffSel:BOOL;
	
	
	rectoVersoInd:BOOL;
	endRollInd:BOOL;
	
	bStartUpBit:BOOL		:= FALSE;
	bStartUp_ResetBit:BOOL	:= FALSE;
	bStartUp_SetBit:BOOL:= FALSE;
	
	SR_RunTimeLimit:	SR;
	
	fbResetRunTimeLimit: TON;
	
	mainDriveOndel: TON;
	
//	bEnableUnwindLift:BOOL	;
//	bEnableRewindLift:BOOL	;
	
	bUnwindCouplingLift	:BOOL	;
	bRewindCouplingLift	:BOOL	;
	
	
	bPrintingOn_q:BOOL;
	bInkingOn_q:BOOL;
	
	
	bCounterReached_i:BOOL;
	bFD1_q:BOOL;
	//bFD2_q:BOOL;
	//bFD3_q:BOOL;
	//bFD4_q:BOOL;
	bFD5_q:BOOL;
	bFD6_q:BOOL;
	//bEXH_q:BOOL;
	
	bEnableUnwindLift2:BOOL;
	bEnableRewindLift2:BOOL;
	//bResetSpeed_q:BOOL;
	bIR9_q:BOOL;
	bEndOfRoll_Calc_gb:BOOL;
	bEndOfRoll_Reached:BOOL;
	
	adiDIAM_MEASUREMENTS:ARRAY[1..10] OF DINT;
	d_mp:DINT:=0;

END_VAR

// MyController/Application/GVL_ENCODER
VAR_GLOBAL
	
	rVitesseRPM_Filt:REAL;
	
	fbTP_STARTUP: TP;

    (* Validity of the capture register value read by the EXPERTGetCapturedValue Function Block: OK (TRUE) or Unknown (FALSE) *)
	bS_Rst:BOOL;
	tStartUp_Time:TIME;
	diFrequency_RAW:DINT;
	
	(*MECHANICAL PARAMETER*)
	
	rInchPerTurn: REAL	:= 12.0;
	rGearBx: REAL		:= 1.5;


	(*USED FOR THE COUNTER*)
	BASE_FINAL_CNT:DINT;
	rInchPerMin:REAL;
	rInchActualCount:REAL;
	rFeetActualCount:REAL;
	
	bUnwindPID_ON_gb:BOOL;
	bUnwindHold_ON_gb:BOOL;

END_VAR

// MyController/Application/GVL_NOT_USED_IOs
VAR_GLOBAL
	
	bVerso1_i :BOOL;
	bRecto1_i :BOOL;
	bVerso2_i :BOOL;
	bRecto2_i: BOOL;

	bANX_RECTO1_q: BOOL;
	bANX_VERSO1_q: BOOL;
	bANX_RECTO2_q: BOOL;
	bANX_VERSO2_q: BOOL;
	
	bInkingOn_i:BOOL;
	bPrintingOn_i:BOOL;
	InkingOn_i:BOOL;
	PrintingOn_i:BOOL;
	bWebBreak_i:BOOL;
	
	bUnwindCoupling_i:BOOL;
	bEnableUnwindLift_i:BOOL;
	bEnableRewindLift_i:BOOL;
	
	bHotMelt_q:BOOL;
	

	//bIR9_q:BOOL;
	bIR10_q:BOOL;
	
	bWasteBlower_q:BOOL;
bFD_Motion5_i:BOOL;	
bFD_Motion6_i:BOOL;
	
	
END_VAR

// MyController/Application/GVL_HMI
VAR_GLOBAL
	
		//TEMPORAIRE POUR LE PROBLEME DE STATION 1
		
		HMI_FLEXO1_bAniloxMtr:BOOL			:= FALSE;
		HMI_FLEXO1_bAniloxKickOff:BOOL 		:= FALSE;
		HMI_FLEXO1_bPlateKickoff:BOOL 		:= FALSE;
		HMI_FLEXO1_bInfraRed:BOOL 			:= FALSE;
		HMI_FLEXO1_bRegAdvance:BOOL			:= FALSE;
		HMI_FLEXO1_bRegRetard:BOOL			:= FALSE;
		HMI_FLEXO1_bRunPlus:BOOL			:= FALSE;
		HMI_FLEXO1_bRunMinus:BOOL			:= FALSE;
		HMI_FLEXO1_bJog:BOOL				:= FALSE;
		HMI_FLEXO1_bStop:BOOL				:= FALSE;
		HMI_FLEXO1_bSetup:BOOL				:= FALSE;
		HMI_FLEXO1_bInkingOn:BOOL			:= FALSE;
		HMI_FLEXO1_bPrintingOn:BOOL			:= FALSE;
		HMI_FLEXO1_bUnlock_i:BOOL			:= FALSE;
		HMI_FLEXO1_bSpare2:BOOL				:= FALSE;
		HMI_FLEXO1_bSpare3:BOOL				:= FALSE;

		
		HMI_FLEXO1_bGreenLight_q:BOOL			:=FALSE;
		HMI_FLEXO1_bArAniloxMotor_KEEP:BOOL		:=FALSE;
		HMI_FLEXO1_bArAniloxKickoff_KEEP:BOOL	:=FALSE;
		HMI_FLEXO1_bArPlateKickoff_KEEP:BOOL	:=FALSE;
		HMI_FLEXO1_bArIR_KEEP:BOOL				:=FALSE;
		HMI_FLEXO1_bArSETUP_KEEP:BOOL			:=FALSE;
		HMI_FLEXO1_bInkingOn_KEEP:BOOL			:=FALSE;
		HMI_FLEXO1_bPrintingOn_KEEP:BOOL		:=FALSE;
		HMI_FLEXO1_bDrawLock_q:BOOL				:=FALSE;
		HMI_FLEXO1_bSpare2_q:BOOL				:=FALSE;
		HMI_FLEXO1_bSpare3_q:BOOL				:=FALSE;
		HMI_FLEXO1_readyInd:BOOL				:=FALSE;
		//


		tempInReal: REAL;
		
		bAniloxOn_Temp:BOOL:=FALSE;
		
		jogPb:BOOL;
		
		bBlowerSel_HMI:BOOL;
		
		bIR1_Low_HMI	:BOOL	:= TRUE;
		bIR1_High_HMI	:BOOL	:= FALSE;
		bIR2_Low_HMI	:BOOL	:= TRUE;
		bIR2_High_HMI	:BOOL	:= FALSE;
		
		bInfeedOnPb_HMI_i	:BOOL;
		bRewindOnPb_HMI_i	:BOOL;
		bTopRewindOnPb_HMI_i	:BOOL;
		bGravureOnPb_HMI_i	:BOOL;
		
		bRollEndOnPb_HMI_i		:BOOL;
		infeedOnOut:BOOL;
		rewindOnOut:BOOL;
		top_rewindOnOut:BOOL;
		gravureOnOut: BOOL;
		aniloxOnOut:BOOL;
		
		slowrotationOnOut:BOOL;
		
		rollendOnOut:BOOL:=0;
		uiRollEndState:UINT:=0;
		bRollEndDetected_HMI:BOOL	:= FALSE;
		okToRun: BOOL;
		
		(*REGISTERS SCREEN*)
		bRegAdvance_1_HMI	:BOOL;
		bRegRetard_1_HMI	:BOOL;
		bRegAdvance_2_HMI	:BOOL;
		bRegRetard_2_HMI	:BOOL;
		bRegAdvance_3_HMI	:BOOL;
		bRegRetard_3_HMI	:BOOL;
		bRegAdvance_4_HMI	:BOOL;
		bRegRetard_4_HMI	:BOOL;
		bRegAdvance_5_HMI	:BOOL;
		bRegRetard_5_HMI	:BOOL;
		bRegAdvance_6_HMI	:BOOL;
		bRegRetard_6_HMI	:BOOL;
		bRegAdvance_7_HMI	:BOOL;
		bRegRetard_7_HMI	:BOOL;
		bRegAdvance_8_HMI	:BOOL;
		bRegRetard_8_HMI	:BOOL;
		bRegAdvance_9_HMI	:BOOL;
		bRegRetard_9_HMI	:BOOL;
		bRegAdvance_10_HMI	:BOOL;
		bRegRetard_10_HMI	:BOOL;
		bRegAdvance_11_HMI	:BOOL;
		bRegRetard_11_HMI	:BOOL;
		bRegAdvance_12_HMI	:BOOL;
		bRegRetard_12_HMI	:BOOL;
		
		bRegAdvance_13_HMI	:BOOL;
		bRegRetard_13_HMI	:BOOL;
		bRegAdvance_14_HMI	:BOOL;
		bRegRetard_14_HMI	:BOOL;
		bRegAdvance_15_HMI	:BOOL;
		bRegRetard_15_HMI	:BOOL;
		bRegAdvance_16_HMI	:BOOL;
		bRegRetard_16_HMI	:BOOL;
		
		bRollEndReset_HMI	:BOOL;
		(*DRYING STATE 1*)
		
		
									
												
		
		
		
		(*MACHINE INTERLOCKS*)
		bEmergencyBeacon_HMI_q:BOOL;
		
		bEndOfRollBeacon_HMI_q:BOOL;
		bAtCountBeacon_HMI_q:BOOL;
		bSafetyGuard_HMI_q:BOOL;
		bCounterReached_HMI_q:BOOL;
		bUnwindCoupling_HMI_q:BOOL;
		bRewindCoupling_HMI_q:BOOL;
		
		bUnwindLiftArm_HMI_q:BOOL;
		bRewindLiftArm_HMI_q:BOOL;
		bReversibleGearBox1_HMI_q:BOOL;
		bReversibleGearBox2_HMI_q:BOOL;
		
		
		(* ACTIVATE SENSORS*)
		
		bUnwindCouplingOn_HMI_i:BOOL;
		bRewindCouplingOn_HMI_i:BOOL;
		bUnwindLiftArmOn_HMI_i:BOOL;
		bRewindLiftArmOn_HMI_i:BOOL;
		
		bSafetyGuardOn_HMI_i:BOOL;
		bWebBreakOn_HMI_i:BOOL;
		
		
		
		
		
	
		(*MACHINE FAULTS*)
		
		(*DRIVE ERRORS*)
		bInfeedDriveTripped_HMI_q:BOOL;
		bRewindDriveTripped_HMI_q:BOOL;
		bAniloxDriveTripped_HMI_q:BOOL;
		
	
		
		(*TENSION*)
		bUnwindWebBreak_HMI_q:BOOL;
		bInfeedWebBreak_HMI_q:BOOL;
		bRewindWebBreak_HMI_q:BOOL;
		
		(*BLOWERS*)
		bFD1_HMI_q:BOOL;
		bEX1_HMI_q:BOOL;
		bFD2_HMI_q:BOOL;
		bEX2_HMI_q:BOOL;
		
		bEXH_HMI_q:BOOL;
		
		fbFAULT_BLK_HMI_q: BLINK;
		bFaultBeacon_HMI_q:BOOL;
		
		fbINTERLOCK_BLK_HMI_q: BLINK;
		bInterlocksBeacon_HMI_q:BOOL;
		
		WebCLNIP_OnOut:BOOL;
		
		bAllDrives_ModbusError_HMI:BOOL;
		bRewindRunSignalMissing_HMI:BOOL;
		bInfeedRunSignalMissing_HMI:BOOL;
		
		bInkSpray_HMI:BOOL;
		
		bInkSpray1On_HMI_i	:BOOL	:= FALSE;
		bInkSpray2On_HMI_i	:BOOL	:= FALSE;
		bInkSpray3On_HMI_i	:BOOL	:= FALSE;
		bInkSpray4On_HMI_i	:BOOL	:= FALSE;
		
		bConveyorOn_HMI_i	:BOOL	:= FALSE;
		bInterlocksOk: BOOL;
		
		bComHealthy_gb			:BOOL	:= FALSE;
		bRelayComHealthy_gb		:BOOL	:= FALSE;
		bAllDriveHealthy_HMI_i	: BOOL;
		
		
		
		bMainIR_HMI_i:BOOL	:= FALSE;
		bWebBreak_HMI_q:BOOL := FALSE;
		bRollEnd_HMI_q:BOOL	:= FALSE;
		
		bFaultReset_HMI_i:BOOL;
		
		bBlowerFaultGroup1_HMI_q:BOOL;
		bBlowerFaultGroup2_HMI_q:BOOL;
		bBlowerFaultGroup3_HMI_q:BOOL;
		bBlowerFaultGroup4_HMI_q:BOOL;
		bBlowerFaultGroup5_HMI_q:BOOL;
		bBlowerFaultGroup6_HMI_q:BOOL;
		bExhOVL_HMI_q:BOOL;
		
		bGeneralBlowerFault_HMI_q:BOOL;
	
		
		bComHeartBeat1_CAN_i:BOOL:=TRUE;
		bComHeartBeat2_CAN_i:BOOL:=TRUE;
		bComHeartBeat3_CAN_i:BOOL:=TRUE;
		bComHeartBeat4_CAN_i:BOOL:=TRUE;
		bComHeartBeat5_CAN_i:BOOL:=TRUE;
		bComHeartBeat6_CAN_i:BOOL:=TRUE;
		bComHeartBeat7_CAN_i:BOOL:=TRUE;
		bComHeartBeat8_CAN_i:BOOL:=TRUE;
		bComHeartBeat9_CAN_i:BOOL:=TRUE;
		bComHeartBeat10_CAN_i:BOOL:=TRUE;
		bComHeartBeat11_CAN_i:BOOL:=TRUE;
		bComHeartBeat12_CAN_i:BOOL:=TRUE;
		bComHeartBeat13_CAN_i:BOOL:=TRUE;

		//bComHeartBeat_CAN_i: ARRAY[1..20]OF BOOL;
		
		bComHeartBeatRelay1_CAN_i:BOOL:=TRUE;
		bComHeartBeatRelay2_CAN_i:BOOL:=TRUE;
		bComHeartBeatRelay3_CAN_i:BOOL:=TRUE;
		bComHeartBeatRelay4_CAN_i:BOOL:=TRUE;
		bComHeartBeatRelay5_CAN_i:BOOL:=TRUE;
		bComHeartBeatRelay6_CAN_i:BOOL:=TRUE;
		bComHeartBeatRelay7_CAN_i:BOOL:=TRUE;
		
		bComHeartBeatRelay1_Bypass_CAN_i:BOOL:=TRUE;
		bComHeartBeatRelay2_Bypass_CAN_i:BOOL:=TRUE;
		bComHeartBeatRelay3_Bypass_CAN_i:BOOL:=TRUE;
		bComHeartBeatRelay4_Bypass_CAN_i:BOOL:=TRUE;
		bComHeartBeatRelay5_Bypass_CAN_i:BOOL:=TRUE;
		bComHeartBeatRelay6_Bypass_CAN_i:BOOL:=TRUE;
		bComHeartBeatRelay7_Bypass_CAN_i:BOOL:=TRUE;
		
		bComHeartBeat1_Bypass_CAN_i	:BOOL:= FALSE;
		bComHeartBeat2_Bypass_CAN_i	:BOOL:= FALSE;
		bComHeartBeat3_Bypass_CAN_i	:BOOL:= FALSE;
		bComHeartBeat4_Bypass_CAN_i	:BOOL:= FALSE;
		bComHeartBeat5_Bypass_CAN_i	:BOOL:= FALSE;
		bComHeartBeat6_Bypass_CAN_i	:BOOL:= FALSE;
		bComHeartBeat7_Bypass_CAN_i	:BOOL:= FALSE;
		bComHeartBeat8_Bypass_CAN_i	:BOOL:= FALSE;
		bComHeartBeat9_Bypass_CAN_i	:BOOL:= FALSE;
		bComHeartBeat10_Bypass_CAN_i	:BOOL:= FALSE;
		bComHeartBeat11_Bypass_CAN_i	:BOOL:= FALSE;
		bComHeartBeat12_Bypass_CAN_i	:BOOL:= FALSE;
		bComHeartBeat13_Bypass_CAN_i	:BOOL:= FALSE;
		
		bComHeartBeat1_HMI_i:BOOL;
		bComHeartBeat2_HMI_i:BOOL;
		bComHeartBeat3_HMI_i:BOOL;
		bComHeartBeat4_HMI_i:BOOL;
		bComHeartBeat5_HMI_i:BOOL;
		bComHeartBeat6_HMI_i:BOOL;
		bComHeartBeat7_HMI_i:BOOL;
		bComHeartBeat8_HMI_i:BOOL;
		bComHeartBeat9_HMI_i:BOOL;
		bComHeartBeat10_HMI_i:BOOL;
		bComHeartBeat11_HMI_i:BOOL;
		bComHeartBeat12_HMI_i:BOOL;
		bComHeartBeat13_HMI_i:BOOL;
		
		
		bComHeartBeatRelay1_HMI_i:BOOL;
		bComHeartBeatRelay2_HMI_i:BOOL;
		bComHeartBeatRelay3_HMI_i:BOOL;
		bComHeartBeatRelay4_HMI_i:BOOL;
		bComHeartBeatRelay5_HMI_i:BOOL;
		bComHeartBeatRelay6_HMI_i:BOOL;
		bComHeartBeatRelay7_HMI_i:BOOL;
		
		
		stDryingGroup_1_HMI_i:stDryingGroup:=(bDryOff_i:=TRUE,bBlowerOn_i:=FALSE,bLowHeatOn_i:=FALSE,bHighHeatOn_i:=FALSE);
												
												
		stDryingGroup_2_HMI_i:stDryingGroup:=(bDryOff_i:=TRUE,bBlowerOn_i:=FALSE,bLowHeatOn_i:=FALSE,bHighHeatOn_i:=FALSE);																				
											
		stDryingGroup_3_HMI_i:stDryingGroup:=(bDryOff_i:=TRUE,bBlowerOn_i:=FALSE,bLowHeatOn_i:=FALSE,bHighHeatOn_i:=FALSE);
		
		stDryingGroup_4_HMI_i:stDryingGroup:=(bDryOff_i:=TRUE,bBlowerOn_i:=FALSE,bLowHeatOn_i:=FALSE,bHighHeatOn_i:=FALSE);
		
		stDryingGroup_5_HMI_i:stDryingGroup:=(bDryOff_i:=TRUE,bBlowerOn_i:=FALSE,bLowHeatOn_i:=FALSE,bHighHeatOn_i:=FALSE);
		
		stDryingGroup_6_HMI_i:stDryingGroup:=(bDryOff_i:=TRUE,bBlowerOn_i:=FALSE,bLowHeatOn_i:=FALSE,bHighHeatOn_i:=FALSE);
		
		stDryingGroup_7_HMI_i:stDryingGroup:=(bDryOff_i:=TRUE,bBlowerOn_i:=FALSE,bLowHeatOn_i:=FALSE,bHighHeatOn_i:=FALSE);
		
		stDryingGroup_8_HMI_i:stDryingGroup:=(bDryOff_i:=TRUE,bBlowerOn_i:=FALSE,bLowHeatOn_i:=FALSE,bHighHeatOn_i:=FALSE);
		
		stDryingGroup_9_HMI_i:stDryingGroup:=(bDryOff_i:=TRUE,bBlowerOn_i:=FALSE,bLowHeatOn_i:=FALSE,bHighHeatOn_i:=FALSE);
		
		stDryingGroup_10_HMI_i:stDryingGroup:=(bDryOff_i:=TRUE,bBlowerOn_i:=FALSE,bLowHeatOn_i:=FALSE,bHighHeatOn_i:=FALSE);
		
		bGravureNipPb_HMI_q:BOOL;
	
		
		bGravureSetup_HMI:BOOL;
		bHotMeltOnOff_HMI:BOOL;
		
		iPlateTimeDelay_HMI:INT:=2;
		tPlateTimeDelay_HMI:TIME:=T#2.0S;
		
		bEmergency_KEEP :BOOL;
		
		bInkingOn_HMI_i:BOOL;
		bPrintingOn_HMI_i:BOOL;
		
		bInkingOn_HMI_q:BOOL;
		bPrintingOn_HMI_q:BOOL;

	bGravure_Tens_Inc_HMI_i:BOOL;
	bGravure_Tens_Dec_HMI_i:BOOL;
	
	bGravure_Reg_Adv_HMI_i:BOOL;
	bGravure_Reg_Ret_HMI_i:BOOL;
	
	bGravure_Jog_Adv_HMI_i:BOOL;
	bGravure_Jog_Ret_HMI_i:BOOL;
	wRexrothCmd_GR_q:WORD;
	wRexrothStatus_GR_i:WORD;
	
	uiGravureRegisterOffset:UINT;
	uiGravureGearingAdjust:UINT;

	uiAccessCode: UINT:= 0;
	bAccessGranted: BOOL:= FALSE;	

	//Status	
	bGravure_StatusDisabled_HMI_q	:BOOL;
	bGravure_StatusSlowRot_HMI_q	:BOOL;
	bGravure_StatusSynch_HMI_q		:BOOL;
	bGravure_StatusError_HMI_q		:BOOL;
	bGravure_StatusLock_HMI_q		:BOOL;
	

	
	bGravure_ResetDrive_HMI_i		:BOOL;
	bGravure_SlwRotate_HMI_i		:BOOL;
	bGravure_Oscillation_HMI_i		:BOOL;
	bGravure_RegiCtrlOn_HMI_i		:BOOL;
	bInfeed_RegiCtrlOn_HMI_i		:BOOL;
	uiGravure_LockPosition_HMI_q	:UINT;		//THIS IS DEFINED IN DEGREES
	uiGravure_Deviation_HMI_q		:UINT;		//THIS IS DEFINED IN DEGREES
	
//	bGravure_DrvReset_HMI_i			:BOOL;

	//This is the deviation between probe mark and the encoder
	rDeviation_HMI_q:REAL;
	rRegiCtrlSetpoint_HMI_q:REAL;
	//This represents the adjustment steps in mil.
	rRegAdjustStep_HMI_i:REAL;
	
	rFPM_HMI_q:REAL;
	
	
	bCounterOn_HMI_i:BOOL;
	bTotCounterOn_HMI_i:BOOL;
	bResetCount_HMI_i:BOOL;
	bTotResetCount_HMI_i:BOOL;
	
	(*ACTUAL COUNTS*)
	rRepeatCount_HMI_q:REAL;
	rRepeatTotCount_HMI_q:REAL;
	diUnwindActualDiam_HMI_q:DINT;
	
	uiUnwindTensDisplay_HMI_q:UINT;
	uiUnwindBrakeOutput_HMI_q:UINT:=0;
	bUnwindManualMode_HMI_i:BOOL;

	
	uiCOUNT_BASE					: UINT:=150;
	bCOUNT_ON_HMI_i					:BOOL:= FALSE;
	bRESET_COUNT_HMI_i				:BOOL:= FALSE;
	bTOTCOUNT_ON_HMI_i				:BOOL:= FALSE;
	bRESET_TOT_COUNT_HMI_i			:BOOL:= FALSE;
	rRAW_TOT_COUNT_BUFFER:REAL;
	rRAW_COUNT_BUFFER:REAL;
	
	
	bInfeed_Tens_Inc_HMI_i			:BOOL;
	bInfeed_Tens_dec_HMI_i			:BOOL;
	bInfeed_ResetDrive_HMI_i		:BOOL;
	bInfeed_Manual_i				:BOOL;
	bInfeed_StatusError_HMI_q		:BOOL;
	bInfeed_StatusDisabled_q		:BOOL;
	bInfeed_StatusSynch_HMI_q		:BOOL;
	bInfeed_StatusSlowRot_HMI_q		:BOOL;
	bInfeed_title_q					:BOOL;
	bInfeed_Tension_HMI				:REAL;
	wInfeedManualGearing_HMI_i		:UINT;
	
	stTensionCtrlState_HMI_i: stTensionCtrlState;
END_VAR

VAR_GLOBAL RETAIN
	
	rDesiredCount_HMI_i:REAL;
	
	rRepeat_HMI_i:REAL;
	rLineShaftGBX_HMI_i:REAL;
	
	diUnwindPresetDiam_HMI_i:DINT;
	
	uiUnwindTensSetpoint_HMI_i:UINT:=50;
	uiUnwindTensManual_HMI_i:UINT;
	uiUnwindTensState_HMI_i:UINT;	(*OFF MANUAL AUTO*)
	
END_VAR

// MyController/Application/GVL_ETHERNET
VAR_GLOBAL

	
	
	InfeedModbusError:BOOL := FALSE;
	RewindModbusError:BOOL := FALSE;
	TopRewindModbusError:BOOL := FALSE;
	AniloxModbusError:BOOL	:= FALSE;
	GravureModbusError:BOOL	:= FALSE;

	bRewindHealthy_ETH:BOOL	:= FALSE;
	bRewindActive_ETH:BOOL	:= FALSE;
	
	bTopRewindHealthy_ETH:BOOL	:= FALSE;
	bTopRewindActive_ETH:BOOL	:= FALSE;
	
	bInfeedHealthy_ETH:BOOL	:= FALSE;
	bInfeedActive_ETH:BOOL	:= FALSE;
	
	bAllDrives_ModbusError:	BOOL	:= FALSE;
	bAllDrivesOK_TO_RUN_ETH	: BOOL	:= FALSE;
	
	
END_VAR

// MyController/Application/GVL_KEEP_ARRAY
VAR_GLOBAL

	FB_LATCH_PLATE_1: SR;
	FB_LATCH_PLATE_2: SR;
	FB_LATCH_PLATE_3: SR;
	FB_LATCH_PLATE_4: SR;
	FB_LATCH_PLATE_5: SR;
	FB_LATCH_PLATE_6: SR;
	FB_LATCH_PLATE_7: SR;
	FB_LATCH_PLATE_8: SR;
	FB_LATCH_PLATE_9: SR;
	FB_LATCH_PLATE_10: SR;
	FB_LATCH_PLATE_11: SR;
	FB_LATCH_PLATE_12: SR;
	
	FB_LATCH_PLATE_20: SR;	//GRAVURE
	
	
	
	
	FB_LATCH_ANILOX_1: SR;
	FB_LATCH_ANILOX_2: SR;
	FB_LATCH_ANILOX_3: SR;
	FB_LATCH_ANILOX_4: SR;
	FB_LATCH_ANILOX_5: SR;
	FB_LATCH_ANILOX_6: SR;
	FB_LATCH_ANILOX_7: SR;
	FB_LATCH_ANILOX_8: SR;
	FB_LATCH_ANILOX_9: SR;
	FB_LATCH_ANILOX_10: SR;
	FB_LATCH_ANILOX_11: SR;
	FB_LATCH_ANILOX_12: SR;
	
	
	FB_LATCH_SETUP_1: SR;
	FB_LATCH_SETUP_2: SR;
	FB_LATCH_SETUP_3: SR;
	FB_LATCH_SETUP_4: SR;
	FB_LATCH_SETUP_5: SR;
	FB_LATCH_SETUP_6: SR;
	FB_LATCH_SETUP_7: SR;
	FB_LATCH_SETUP_8: SR;
	FB_LATCH_SETUP_9: SR;
	FB_LATCH_SETUP_10: SR;
	
	FB_LATCH_SETUP_20: SR;	//GRAVURE
	
	
	//bRewindPID_Out:BOOL;
	runOut:BOOL;
	jogOut:BOOL;
	recto1Out:BOOL;
	verso1Out:BOOL;
	recto2Out:BOOL;
	verso2Out:BOOL;
	
	bSetup_KEEP:BOOL;
	bEndOfRoll_KEEP:BOOL;
	readyInd:BOOL;
	
	//*******************************************
	//**  SETUP  			*********************
	//*******************************************
	
	bArSETUP_KEEP:	ARRAY[1..20]OF BOOL;
	
	//*******************************************
	//**  ANILOX CYLINDER	*********************
	//*******************************************

	bAniloxKickoffEnable_KEEP	:BOOL 	:= FALSE;
	bArAniloxKickoff_KEEP:	ARRAY[1..20]OF BOOL;
	fbArAniloxKickoff_KEEP:	ARRAY[1..20]OF SR;
	
	bArAniloxKickoff_Enable_KEEP	:	ARRAY[1..20]OF BOOL;
	
	bAniloxKickoff_q:	ARRAY[1..20]OF BOOL;	//OUTPUT

	//*******************************************
	//**  PLATE CYLINDER	*********************
	//*******************************************

	bPlateKickoffEnable_KEEP	:BOOL	:= FALSE;
	bArPlateKickoff_Enable_KEEP	:	ARRAY[1..20]OF BOOL;

	bArPlateKickoff_KEEP:	ARRAY[1..20]OF BOOL;
	fbArPlateKickoff_KEEP:	ARRAY[1..20]OF SR;
	
	bPlateKickoff_q:	ARRAY[1..20]OF BOOL;	//OUTPUT
	
	
	bInkingOn_KEEP:BOOL:=FALSE;
	bPrintingOn_KEEP:BOOL:=FALSE;
	//bPrintingOn_q: BOOL;
	
	bArAniloxMotor_KEEP:	ARRAY[1..20]OF BOOL;
	fbArAniloxMotor_KEEP:	ARRAY[1..20]OF SR;
	
	bArIR_KEEP:				ARRAY[1..20]OF BOOL;
	
	bWasteBlower_KEEP:BOOL;	
//bIR1_KEEP:BOOL	:= FALSE;
	//bIR2_KEEP:BOOL	:= FALSE;
	//bIR3_KEEP:BOOL	:= FALSE;
	//bIR4_KEEP:BOOL	:= FALSE;
	
	
	
	SR_RollEnd_KEEP:SR;
	SR_RollEndDetect_KEEP:SR;
	
	FB_IR1_KEEP:SR;
	FB_IR2_KEEP:SR;
	FB_IR3_KEEP:SR;
	FB_IR4_KEEP:SR;
	FB_IR5_KEEP:SR;
	FB_IR6_KEEP:SR;
	FB_IR7_KEEP:SR;
	FB_IR8_KEEP:SR;
	FB_IR9_KEEP:SR;
	FB_IR10_KEEP:SR;

	FB_WasteBlower_KEEP:SR;
	
	fbRUNOUT_REAL:TON;
	
	
END_VAR

// MyController/Application/GVL_CONVERT
VAR_GLOBAL


//Application.ArFlexoStation[1].bAniloxMot_q
//Application.GVL_CAN_ARRAY.ArFlexoStation[1].bPlateKickoff_q
//Application.GVL_CAN_ARRAY.ArFlexoStation[1].bRegAdvance_q


bAnxMot_q1	:BOOL;
bAnxMot_q2	:BOOL;
bAnxMot_q3	:BOOL;
bAnxMot_q4	:BOOL;
bAnxMot_q5	:BOOL;
bAnxMot_q6	:BOOL;
bAnxMot_q7	:BOOL;
bAnxMot_q8	:BOOL;
bAnxMot_q9	:BOOL;
bAnxMot_q10	:BOOL;

bPlateKickoff_q1 :BOOL;
bPlateKickoff_q2 :BOOL;
bPlateKickoff_q3 :BOOL;
bPlateKickoff_q4 :BOOL;
bPlateKickoff_q5 :BOOL;
bPlateKickoff_q6 :BOOL;
bPlateKickoff_q7 :BOOL;
bPlateKickoff_q8 :BOOL;
bPlateKickoff_q9 :BOOL;
bPlateKickoff_q10 :BOOL;

bAnxKickoff_q1 :BOOL;
bAnxKickoff_q2 :BOOL;
bAnxKickoff_q3 :BOOL;
bAnxKickoff_q4 :BOOL;
bAnxKickoff_q5 :BOOL;
bAnxKickoff_q6 :BOOL;
bAnxKickoff_q7 :BOOL;
bAnxKickoff_q8 :BOOL;
bAnxKickoff_q9 :BOOL;
bAnxKickoff_q10 :BOOL;

bRegAdv_q1	:BOOL;
bRegAdv_q2	:BOOL;
bRegAdv_q3	:BOOL;
bRegAdv_q4	:BOOL;
bRegAdv_q5	:BOOL;
bRegAdv_q6	:BOOL;
bRegAdv_q7	:BOOL;
bRegAdv_q8	:BOOL;
bRegAdv_q9	:BOOL;
bRegAdv_q10	:BOOL;


bRegRet_q1	:BOOL;
bRegRet_q2	:BOOL;
bRegRet_q3	:BOOL;
bRegRet_q4	:BOOL;
bRegRet_q5	:BOOL;
bRegRet_q6	:BOOL;
bRegRet_q7	:BOOL;
bRegRet_q8	:BOOL;
bRegRet_q9	:BOOL;
bRegRet_q10	:BOOL;



END_VAR

// MyController/Application/GVL_KEY
VAR_GLOBAL
	
	(*KEYPAD STATION 1*)
	(*KEY DEFINITION*)
	bAniloxMtr_1	: BOOL := FALSE;
	bAniloxKickOff_1	: BOOL := FALSE;
	bPlateKickoff_1	: BOOL := FALSE;
	bInfraRed_1		: BOOL := FALSE;
	bRegAdvance_1	: BOOL	:= FALSE;
	bRegRetard_1		: BOOL	:= FALSE;
	bRunPlus_1		: BOOL	:= FALSE;
	bRunMinus_1		: BOOL	:= FALSE;
	bJog_1			: BOOL	:= FALSE;
	bStop_1			: BOOL	:= FALSE;
	bPrintingOn_1	:BOOL	:= FALSE;
	bInkingOn_1		:BOOL	:= FALSE;
	bSetup_1		:BOOL	:= FALSE;
	bSpare1_1		:BOOL	:= FALSE;
	bSpare2_1		:BOOL	:= FALSE;
	bSpare3_1		:BOOL	:= FALSE;
	
	(*LED DEFINITION*)
	bAniloxMtr_1_LED_q		: BOOL := FALSE;
	bAniloxKickOff_1_LED_q	: BOOL := FALSE;
	bPlateKickoff_1_LED_q	: BOOL := FALSE;
	bInfraRed_1_LED_q		: BOOL := FALSE;
	(*bRun_1_LED_q		: BOOL	:= FALSE;*)
	(*bRegRetard_1_LED_q		: BOOL	:= FALSE;*)
	
	

	(*KEYPAD STATION 2*)
	bAniloxMtr_2	: BOOL := FALSE;
	bAniloxKickOff_2	: BOOL := FALSE;
	bPlateKickoff_2	: BOOL := FALSE;
	bInfraRed_2		: BOOL := FALSE;
	bRegAdvance_2	: BOOL	:= FALSE;
	bRegRetard_2		: BOOL	:= FALSE;
	bRunPlus_2		: BOOL	:= FALSE;
	bRunMinus_2		: BOOL	:= FALSE;
	bJog_2			: BOOL	:= FALSE;
	bStop_2			: BOOL	:= FALSE;
	bPrintingOn_2	:BOOL	:= FALSE;
	bInkingOn_2		:BOOL	:= FALSE;
	bSetup_2		:BOOL	:= FALSE;
	
	
	(*KEYPAD STATION 3*)
	bAniloxMtr_3	: BOOL := FALSE;
	bAniloxKickOff_3	: BOOL := FALSE;
	bPlateKickoff_3	: BOOL := FALSE;
	bInfraRed_3		: BOOL := FALSE;
	bRegAdvance_3	: BOOL	:= FALSE;
	bRegRetard_3		: BOOL	:= FALSE;
	bRunPlus_3		: BOOL	:= FALSE;
	bRunMinus_3		: BOOL	:= FALSE;
	bJog_3			: BOOL	:= FALSE;
	bStop_3			: BOOL	:= FALSE;
	bPrintingOn_3	:BOOL	:= FALSE;
	bInkingOn_3		:BOOL	:= FALSE;
	bSetup_3		:BOOL	:= FALSE;
	

	(*KEYPAD STATION 4*)
	bAniloxMtr_4	: BOOL := FALSE;
	bAniloxKickOff_4	: BOOL := FALSE;
	bPlateKickoff_4	: BOOL := FALSE;
	bInfraRed_4		: BOOL := FALSE;
	bRegAdvance_4	: BOOL	:= FALSE;
	bRegRetard_4		: BOOL	:= FALSE;
	bRunPlus_4		: BOOL	:= FALSE;
	bRunMinus_4		: BOOL	:= FALSE;
	bJog_4			: BOOL	:= FALSE;
	bStop_4			: BOOL	:= FALSE;
	bPrintingOn_4	:BOOL	:= FALSE;
	bInkingOn_4		:BOOL	:= FALSE;
	bSetup_4		:BOOL	:= FALSE;
	
	
	(*KEYPAD STATION 5*)
	bAniloxMtr_5	: BOOL := FALSE;
	bAniloxKickOff_5	: BOOL := FALSE;
	bPlateKickoff_5	: BOOL := FALSE;
	bInfraRed_5		: BOOL := FALSE;
	bRegAdvance_5	: BOOL	:= FALSE;
	bRegRetard_5		: BOOL	:= FALSE;
	bRunPlus_5		: BOOL	:= FALSE;
	bRunMinus_5		: BOOL	:= FALSE;
	bJog_5			: BOOL	:= FALSE;
	bStop_5			: BOOL	:= FALSE;
	bPrintingOn_5	:BOOL	:= FALSE;
	bInkingOn_5		:BOOL	:= FALSE;
	bSetup_5		:BOOL	:= FALSE;
	
END_VAR

// MyController/Application/GVL_DEBUG
VAR_GLOBAL


	
	bComHasFailed_CAN: BOOL := FALSE;
	bComHasFailed_ETH: BOOL := FALSE;
	
	bGbx1_Error: BOOL;
	bGbx2_Error: BOOL;
	
	


END_VAR

// MyController/Application/GVL_counter
VAR_GLOBAL
	
GVL_diff:DINT:=0;
UW_Nbr_Pulses:DINT;
	diNbr_Pulses_FILT: DINT;
	diDIFFERENCE:DINT:=0;
	diDIFFERENCE_Filt:DINT;
	bUW_Flag :BOOL := FALSE;
	
	diCurrentValue:DINT:=10000;
	diLatchedValue:DINT;
	diOldValue:DINT;
	diOLD_VALUE:DINT;
END_VAR

// MyController/Application/COUNTER/PLC_PRG_LD_1
PROGRAM PLC_PRG_LD_1
VAR

TOTAL:DINT;
NEW_VALUE:DINT;
OLD_VALUE:DINT;
INIT:BOOL:=FALSE;
  
CAP_FLAG:BOOL;
    (**********************************************)
    (* HSC Main One-Shot Variables (HSCMain_M258) *)
    (**********************************************)

    (* HSC Input: Forced Enable --> User command *)
    v_xHscMainOneShot_ForcedEnable  : BOOL := FALSE;

    (* HSC Input: Forced Preset --> User command (automatically reset after use) *)
    v_xHscMainOneShot_ForcedPreset  : BOOL := FALSE;

    (* HSC Input: Forced Output0 --> User command *)
    v_xHscMainOneShot_ForcedOutput0 : BOOL := FALSE;

    (* HSC Input: Forced Output1 --> User command *)
    v_xHscMainOneShot_ForcedOutput1 : BOOL := FALSE;

    (* HSC Input: Automatic reset of the "Preset_Flag" output *)
    v_xHscMain_PresetFlag_AutoReset : BOOL := FALSE;

    (* HSC Input: Acknowledgement of the "Captured Value" *)
    v_xHscMain_CapturedValue_Ack    : BOOL := FALSE;

    (* HSC Output: HSC_REF --> Reference to the HSC (for the Administrative Function Blocks) *)
    v_tHscMainOneShot_HSC_REF       : EXPERT_REF := 0;

    (* HSC Output: Error --> TRUE if an error was detected *)
    v_xHscMainOneShot_HSC_Err       : BOOL := FALSE;

    (* HSC Output: Validity --> TRUE if the output values are valid *)
    v_xHscMainOneShot_Validity      : BOOL := TRUE;

    (* Opposite of the "Run" HSC Output: TRUE if the HSC is finished and needs a Rising Edge on its "Sync" input *)
    v_xHscMainOneShot_SYNC_NEEDED   : BOOL := FALSE;

    (* HSC Output: TH0 --> Set to 1 when CurrentValue >= Threshold 0 *)
    v_xHscMainOneShot_GT_TH0        : BOOL := FALSE;

    (* HSC Output: TH1 --> Set to 1 when CurrentValue >= Threshold 1 *)
    v_xHscMainOneShot_GT_TH1        : BOOL := FALSE;

    (* HSC Output: TH2 --> Set to 1 when CurrentValue >= Threshold 2 *)
    v_xHscMainOneShot_GT_TH2        : BOOL := FALSE;

    (* HSC Output: TH3 --> Set to 1 when CurrentValue >= Threshold 3 *)
    v_xHscMainOneShot_GT_TH3        : BOOL := FALSE;

    (* HSC Output: Flag indicating the presence of a new "Captured Value" in the Capture register *)
    v_xHscMain_CapturedValue_Flag   : BOOL := FALSE;

    (* HSC Output: State of Reflex0 *)
    v_xHscMainOneShot_Reflex0       : BOOL := FALSE;

    (* HSC Output: State of Reflex1 *)
    v_xHscMainOneShot_Reflex1       : BOOL := FALSE;

    (* HSC Output: State of physical output Output0 (if Reflex0 configured) *)
    v_xHscMainOneShot_Out0          : BOOL := FALSE;

    (* HSC Output: State of physical output Output1 (if Reflex1 configured) *)
    v_xHscMainOneShot_Out1          : BOOL := FALSE;

    (* HSC Output: CurrentValue --> Current counter value (CV) of the counter *)
    v_xHscMainOneShot_CV            : DINT := 0;


    (*********************************************************)
    (* HSC Main One-Shot Variables (EXPERTGetImmediateValue) *)
    (*********************************************************)

    (* User command to read the HSC Simple counter's current value *)
    v_xCmdGetImmediateValueHscSimple: BOOL := FALSE;

    (* User command to read the HSC Main counter's current value *)
    v_xCmdGetImmediateValueHscMain  : BOOL := FALSE;

    (* EXPERTGetImmediateValue Function Return Value *)
    v_diRetGetImmediateValue        : DINT := 0;

    (* EXPERTGetImmediateValue Function Output: Error --> TRUE if an error was detected *)
    v_xGetImmediateValue_Error      : BOOL := FALSE;

    (* EXPERTGetImmediateValue Function Output: ErrID --> Type of the detected error *)
    v_tGetImmediateValue_ErrID      : EXPERT_IMMEDIATE_ERR_TYPE := EXPERT_IMMEDIATE_ERR_TYPE.EXPERT_IMMEDIATE_FUNC_NO_ERROR;

    (* HSC Simple counter's immediate value, as read by the EXPERTGetImmediateValue Function (-1 for "unknown") *)
    v_diHscSimpleImmediateValue     : DINT := -1;

    (* HSC Main   counter's immediate value, as read by the EXPERTGetImmediateValue Function (-1 for "unknown") *)
    v_diHscMainImmediateValue       : DINT := -1;


    (********************************************************)
    (* HSC Main One-Shot Variables (EXPERTGetCapturedValue) *)
    (********************************************************)

    (* "Execute" input of the EXPERTGetCapturedValue Function Block:                            *)
    (*  - Rising  Edge: Starts the EXPERTGetCapturedValue for the HSC defined by its EXPERT_REF *)
    (*  - Falling Edge: Resets the outputs of this Function Block when it is finished           *)
    v_xEXPERTGetCapturedVal_Execute       : BOOL := FALSE;

    (* Memorization of the value of "v_xEXPERTGetCapturedVal_Execute" *)
    v_xEXPERTGetCapturedVal_Execute_Mem   : BOOL := FALSE;

    (* Flag set to TRUE when the current Get Captured Value operation is finished *)
    v_xEXPERTGetCapturedValIsFinished     : BOOL := FALSE;

    (* Check result of the HSC Reference *)
    v_xEXPERTGetCapturedValRefIsOk        : BOOL := FALSE;

    (* Flag set to TRUE when all conditions for starting a Get Captured Value operation are present *)
    v_xStartGetCapturedValue              : BOOL := FALSE;

    (* "EXPERT_REF_IN" input of the EXPERTGetCapturedValue Function Block: *)
    (* Reference to the HSC; must not be changed during block execution    *)
    v_tEXPERTGetCapturedVal_EXPERT_REF_IN : EXPERT_REF := 0;

    (* "CaptureNumber" input of the EXPERTGetCapturedValue Function Block: Index of the capture register *)
    v_bEXPERTGetCapturedVal_CaptNumber    : BYTE := 0;

    (* EXPERTGetCapturedValue Function Block for returning the contents *)
    (* of one capture register of one principal EXPERT I/O function     *)
    HscMainOneShot_GetCapturedValue       : EXPERTGetCapturedValue;

    (* Value of the capture register of the HSC counter, as read by the EXPERTGetCapturedValue Function Block *)
    v_diHscMainOneShot_CapturedVal        : DINT := 0;

    (* Validity of the capture register value read by the EXPERTGetCapturedValue Function Block: OK (TRUE) or Unknown (FALSE) *)
    v_xHscMainOneShot_GetCaptValOK        : BOOL := FALSE;

    (* Flag set to TRUE when the current Get Captured Value operation is finished AND if the Reference of the read HSC is OK *)
    v_xFlagGetCVFinishedAndRefOK          : BOOL := FALSE;

    (* Flag set to TRUE when the current Get Captured Value operation is successful *)
    v_xGetCVIsSuccessful                  : BOOL := FALSE;

	timer1: TON;
	bZeroSpeed_i: BOOL;
	rVitesseRPM: REAL;
	
	tTIME_BASE:DWORD:=500;
	fbINTEGRAL: STATISTICS_REAL;
	
	bRESET_BLOCK:BOOL:= FALSE;
	bErrorRst: BOOL := false;
	fbFILTER: FILTER_MOVINGAVERAGE;
	
	bFilterBusy_q:BOOL;
	bOutputValid_q:BOOL:= FALSE;
	bFilterError_q:BOOL;
	uiFilterErrorId_q:UINT;
	
	CurrentValue:DINT:=0;
	diff:DINT:=0;
	cache:Dint:=0;
	abc: BOOL:=TRUE;
	def: BOOL:=TRUE;
	indicateur: BOOL;
	timer5: TP;
	bResetTHEBLOCK:BOOL;
	g: BOOL;
	h: BOOL;
	i: BOOL;
	j: BOOL;
	k: BOOL;
	l: BOOL;
	fbTrig: R_TRIG;
	blhldas:bool;
	indicateur2: BOOL;
END_VAR
VAR // added by the converter: edge detectors and wires of the graphical bodies
    _rt1, _rt2 : R_TRIG;
    _w1 : BOOL;
END_VAR

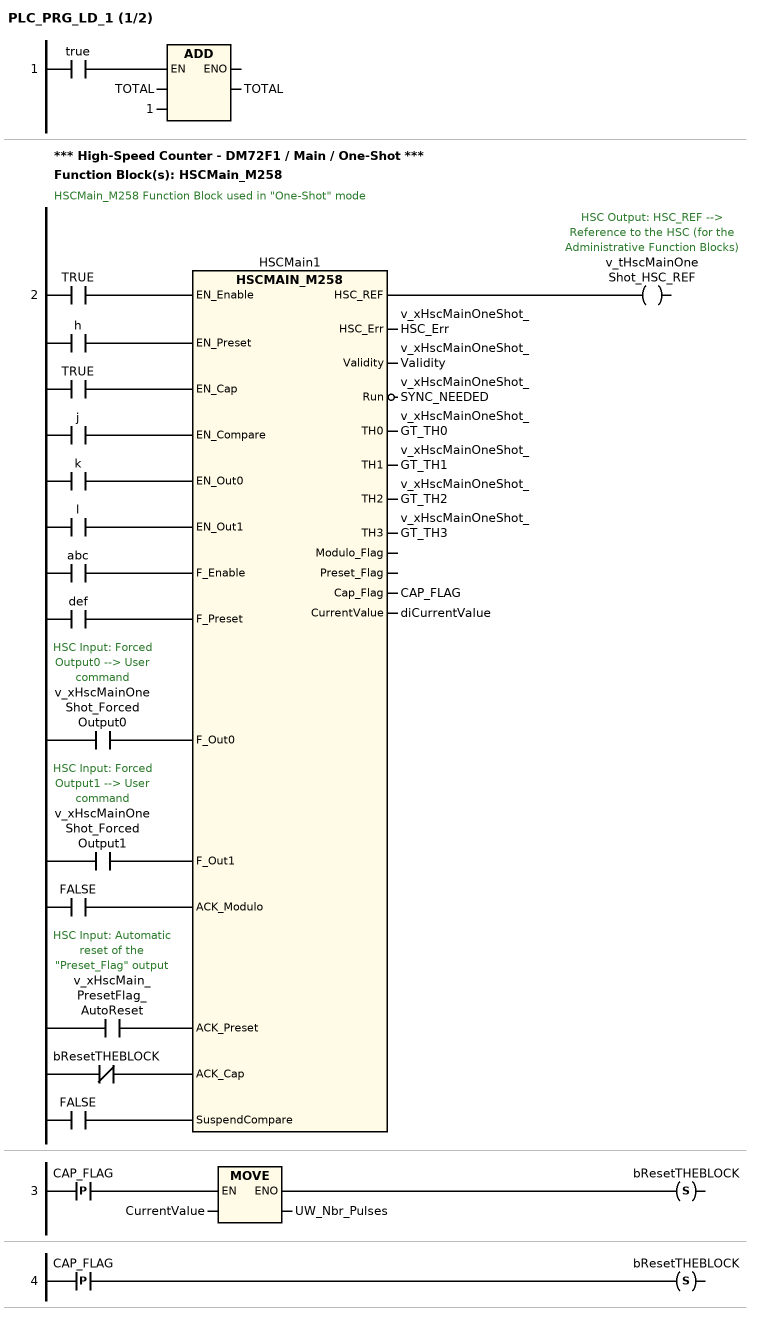
// NETWORK 1
IF true THEN TOTAL := TOTAL + 1; END_IF

// NETWORK 2: *** High-Speed Counter - DM72F1 / Main / One-Shot *** Function Block(s): HSCMain_M258
// HSCMain_M258 Function Block used in "One-Shot" mode
//   v_xHscMainOneShot_ForcedOutput0: HSC Input: Forced Output0 --> User command
//   v_xHscMainOneShot_ForcedOutput1: HSC Input: Forced Output1 --> User command
//   v_xHscMain_PresetFlag_AutoReset: HSC Input: Automatic reset of the "Preset_Flag" output
//   v_xHscMainOneShot_HSC_Err: HSC Output: Error --> TRUE if an error was detected
//   v_xHscMainOneShot_Validity: HSC Output: Validity --> TRUE if the output values are valid
//   v_xHscMainOneShot_GT_TH0: HSC Output: TH0 --> Set to 1 when CurrentValue >= Threshold 0
//   v_xHscMainOneShot_GT_TH1: HSC Output: TH1 --> Set to 1 when CurrentValue >= Threshold 1
//   v_xHscMainOneShot_GT_TH2: HSC Output: TH2 --> Set to 1 when CurrentValue >= Threshold 2
//   v_xHscMainOneShot_GT_TH3: HSC Output: TH3 --> Set to 1 when CurrentValue >= Threshold 3
//   v_xHscMainOneShot_SYNC_NEEDED: Opposite of the "Run" HSC Output: TRUE if the HSC is finished and needs a Rising Edge on its "Sync" input
//   v_tHscMainOneShot_HSC_REF: HSC Output: HSC_REF --> Reference to the HSC (for the Administrative Function Blocks)
HSCMain1(
    EN_Enable := TRUE,
    EN_Preset := h,
    EN_Cap := TRUE,
    EN_Compare := j,
    EN_Out0 := k,
    EN_Out1 := l,
    F_Enable := abc,
    F_Preset := def,
    F_Out0 := v_xHscMainOneShot_ForcedOutput0,
    F_Out1 := v_xHscMainOneShot_ForcedOutput1,
    ACK_Modulo := FALSE,
    ACK_Preset := v_xHscMain_PresetFlag_AutoReset,
    ACK_Cap := NOT bResetTHEBLOCK,
    SuspendCompare := FALSE,
    HSC_Err => v_xHscMainOneShot_HSC_Err,
    Validity => v_xHscMainOneShot_Validity,
    TH0 => v_xHscMainOneShot_GT_TH0,
    TH1 => v_xHscMainOneShot_GT_TH1,
    TH2 => v_xHscMainOneShot_GT_TH2,
    TH3 => v_xHscMainOneShot_GT_TH3,
    Cap_Flag => CAP_FLAG,
    CurrentValue => diCurrentValue); // HSCMAIN_M258
v_xHscMainOneShot_SYNC_NEEDED := NOT HSCMain1.Run;
v_tHscMainOneShot_HSC_REF := HSCMain1.HSC_REF;

// NETWORK 3
_rt1(CLK := CAP_FLAG);
_w1 := _rt1.Q;
IF _w1 THEN UW_Nbr_Pulses := CurrentValue; END_IF
bResetTHEBLOCK S= _w1;

// NETWORK 4
_rt2(CLK := CAP_FLAG);
bResetTHEBLOCK S= _rt2.Q;

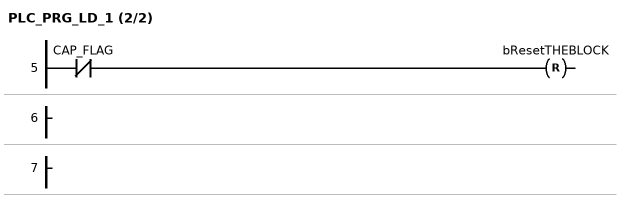
// NETWORK 5
bResetTHEBLOCK R= NOT CAP_FLAG;

// NETWORK 6

// NETWORK 7

END_PROGRAM

// MyController/Application/Main
PROGRAM Main
VAR

	


	
	

	
	
	
	
	SR_WebCleanerOn: 	SR;


	FB_LATCH_WEBCL_STICK: SR;
	bWebCleanerEnable_KEEP: BOOL;
	timerStick: TON;
	
	
	fbRUNOUT: TP;
	fbWebGripperTON: TON;
	FB_LATCH_SETUP_11: SR;
	FB_LATCH_SETUP_12: SR;
END_VAR
VAR_OUTPUT

	
END_VAR
VAR // added by the converter: edge detectors and wires of the graphical bodies
    _rt1, _rt2, _rt3, _rt4, _rt5, _rt6, _rt7, _rt8, _rt9, _rt10, _rt11, _rt12, _rt13, _rt14, _rt15, _rt16, _rt17, _rt18, _rt19, _rt20, _rt21, _rt22, _rt23, _rt24, _rt25, _rt26, _rt27, _rt28, _rt29 : R_TRIG;
    _w1, _w2 : BOOL;
    _ft1, _ft2 : F_TRIG;
END_VAR

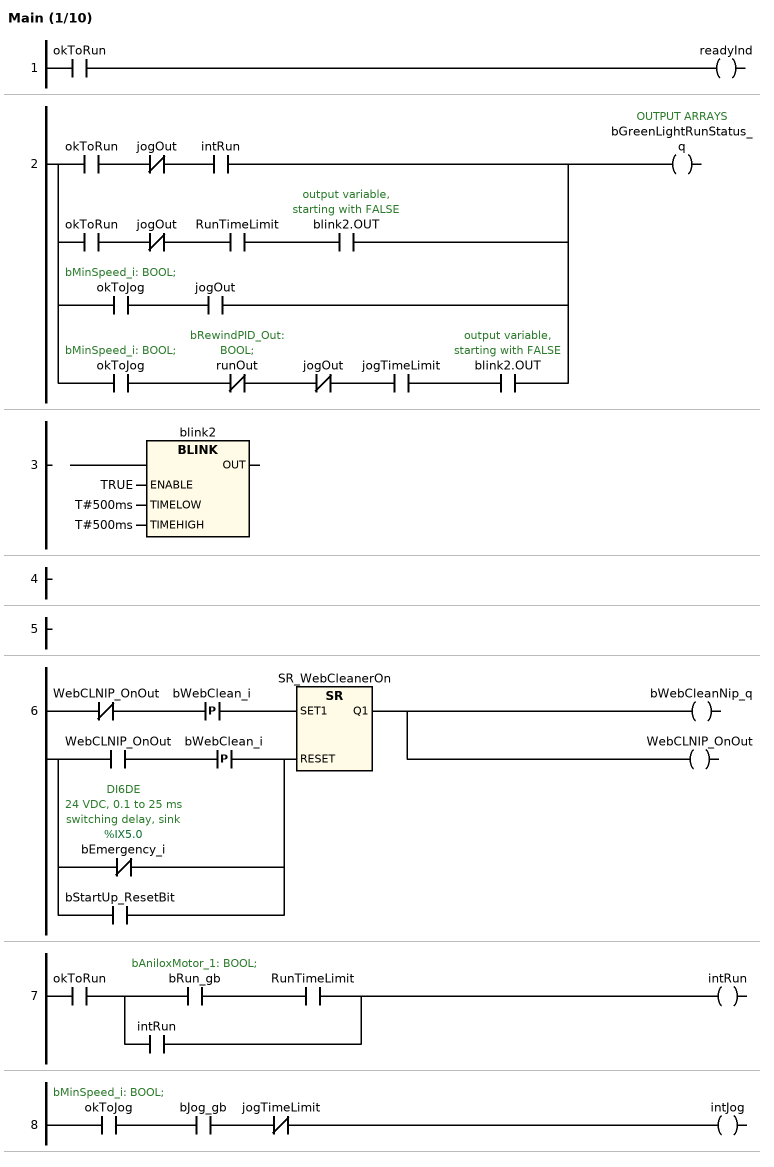
// NETWORK 1
readyInd := okToRun;

// NETWORK 2
//   blink2.OUT: output variable, starting with FALSE
//   okToJog: bMinSpeed_i: BOOL;
//   runOut: bRewindPID_Out:BOOL;
//   bGreenLightRunStatus_q: OUTPUT ARRAYS
bGreenLightRunStatus_q := okToRun AND NOT jogOut AND intRun OR okToRun AND NOT jogOut AND RunTimeLimit AND blink2.OUT OR okToJog AND jogOut OR okToJog AND NOT runOut AND NOT jogOut AND jogTimeLimit AND blink2.OUT;

// NETWORK 3
blink2(ENABLE := TRUE, TIMELOW := T#500ms, TIMEHIGH := T#500ms); // BLINK

// NETWORK 4

// NETWORK 5

// NETWORK 6
//   bEmergency_i: DI6DE 24 VDC, 0.1 to 25 ms switching delay, sink | AT %IX5.0
_rt1(CLK := bWebClean_i);
_rt2(CLK := bWebClean_i);
SR_WebCleanerOn(SET1 := NOT WebCLNIP_OnOut AND _rt1.Q, RESET := WebCLNIP_OnOut AND _rt2.Q OR NOT bEmergency_i OR bStartUp_ResetBit); // SR
bWebCleanNip_q := SR_WebCleanerOn.Q1;
WebCLNIP_OnOut := SR_WebCleanerOn.Q1;

// NETWORK 7
//   bRun_gb: bAniloxMotor_1: BOOL;
intRun := okToRun AND (bRun_gb AND RunTimeLimit OR intRun);

// NETWORK 8
//   okToJog: bMinSpeed_i: BOOL;
intJog := okToJog AND bJog_gb AND NOT jogTimeLimit;

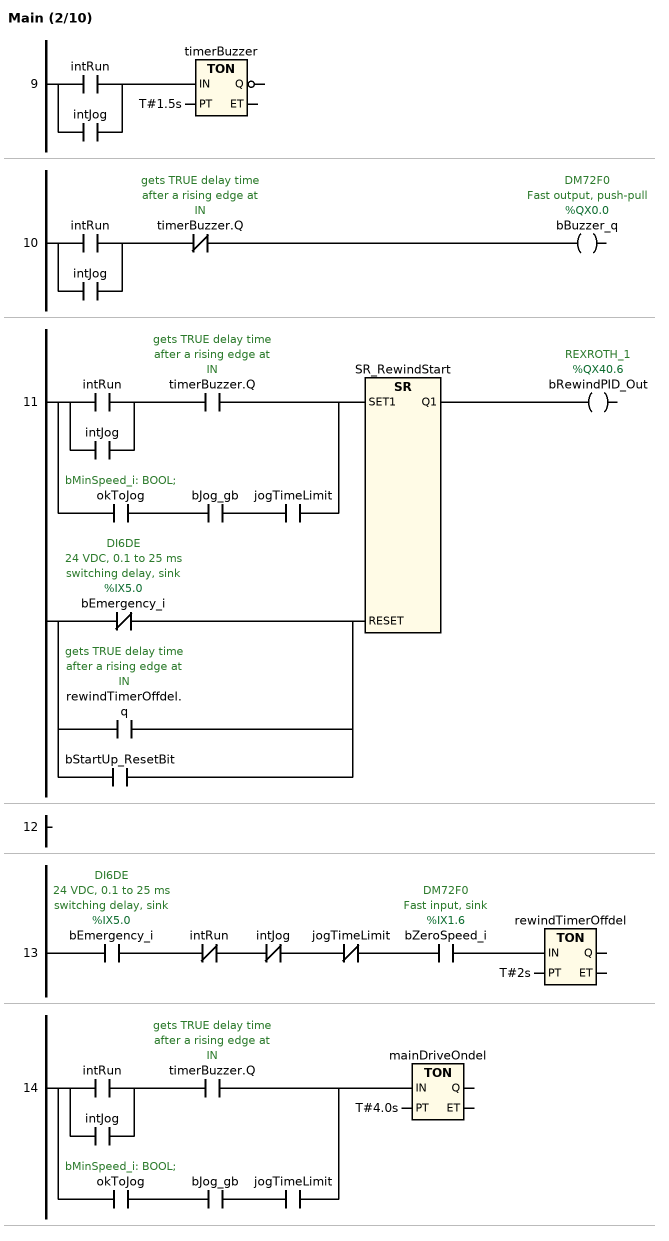
// NETWORK 9
timerBuzzer(IN := intRun OR intJog, PT := T#1.5s); // TON

// NETWORK 10
//   timerBuzzer.Q: gets TRUE delay time after a rising edge at IN
//   bBuzzer_q: DM72F0 Fast output, push-pull | AT %QX0.0
bBuzzer_q := (intRun OR intJog) AND NOT timerBuzzer.Q;

// NETWORK 11
//   timerBuzzer.Q: gets TRUE delay time after a rising edge at IN
//   okToJog: bMinSpeed_i: BOOL;
//   bEmergency_i: DI6DE 24 VDC, 0.1 to 25 ms switching delay, sink | AT %IX5.0
//   rewindTimerOffdel.q: gets TRUE delay time after a rising edge at IN
//   bRewindPID_Out: REXROTH_1 | AT %QX40.6
SR_RewindStart(SET1 := (intRun OR intJog) AND timerBuzzer.Q OR okToJog AND bJog_gb AND jogTimeLimit, RESET := NOT bEmergency_i OR rewindTimerOffdel.q OR bStartUp_ResetBit); // SR
bRewindPID_Out := SR_RewindStart.Q1;

// NETWORK 12

// NETWORK 13
//   bEmergency_i: DI6DE 24 VDC, 0.1 to 25 ms switching delay, sink | AT %IX5.0
//   bZeroSpeed_i: DM72F0 Fast input, sink | AT %IX1.6
rewindTimerOffdel(IN := bEmergency_i AND NOT intRun AND NOT intJog AND NOT jogTimeLimit AND bZeroSpeed_i, PT := T#2s); // TON

// NETWORK 14
//   timerBuzzer.Q: gets TRUE delay time after a rising edge at IN
//   okToJog: bMinSpeed_i: BOOL;
mainDriveOndel(IN := (intRun OR intJog) AND timerBuzzer.Q OR okToJog AND bJog_gb AND jogTimeLimit, PT := T#4.0s); // TON

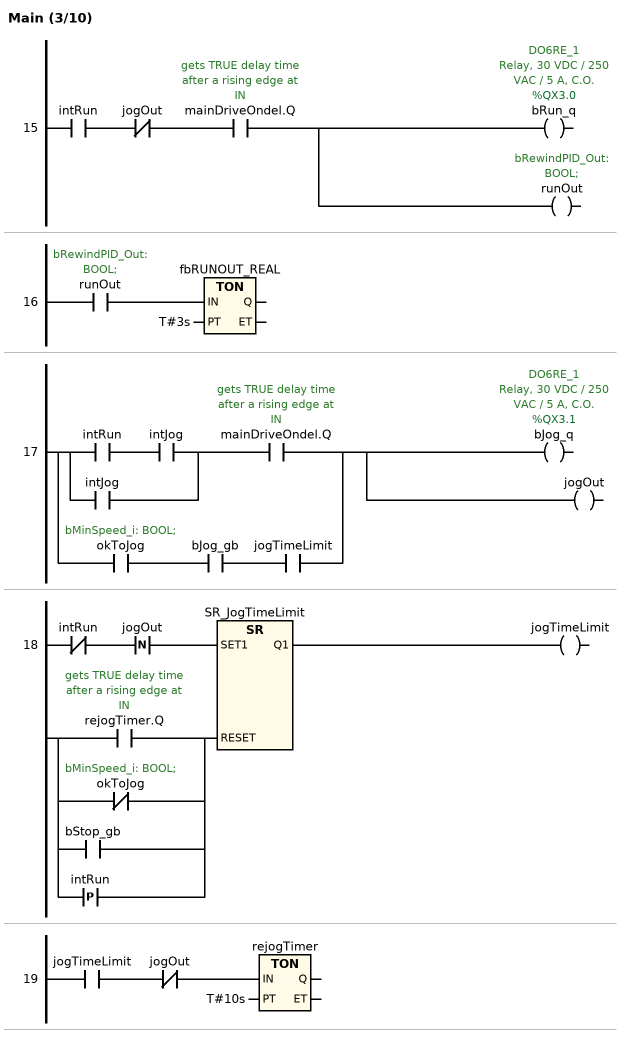
// NETWORK 15
//   mainDriveOndel.Q: gets TRUE delay time after a rising edge at IN
//   bRun_q: DO6RE_1 Relay, 30 VDC / 250 VAC / 5 A, C.O. | AT %QX3.0
//   runOut: bRewindPID_Out:BOOL;
_w1 := intRun AND NOT jogOut AND mainDriveOndel.Q;
bRun_q := _w1;
runOut := _w1;

// NETWORK 16
//   runOut: bRewindPID_Out:BOOL;
fbRUNOUT_REAL(IN := runOut, PT := T#3s); // TON

// NETWORK 17
//   mainDriveOndel.Q: gets TRUE delay time after a rising edge at IN
//   okToJog: bMinSpeed_i: BOOL;
//   bJog_q: DO6RE_1 Relay, 30 VDC / 250 VAC / 5 A, C.O. | AT %QX3.1
_w2 := (intRun AND intJog OR intJog) AND mainDriveOndel.Q OR okToJog AND bJog_gb AND jogTimeLimit;
bJog_q := _w2;
jogOut := _w2;

// NETWORK 18
//   rejogTimer.Q: gets TRUE delay time after a rising edge at IN
//   okToJog: bMinSpeed_i: BOOL;
_ft1(CLK := jogOut);
_rt3(CLK := intRun);
SR_JogTimeLimit(SET1 := NOT intRun AND _ft1.Q, RESET := rejogTimer.Q OR NOT okToJog OR bStop_gb OR _rt3.Q); // SR
jogTimeLimit := SR_JogTimeLimit.Q1;

// NETWORK 19
//   rejogTimer: mainDriveOndel: TON;
rejogTimer(IN := jogTimeLimit AND NOT jogOut, PT := T#10s); // TON

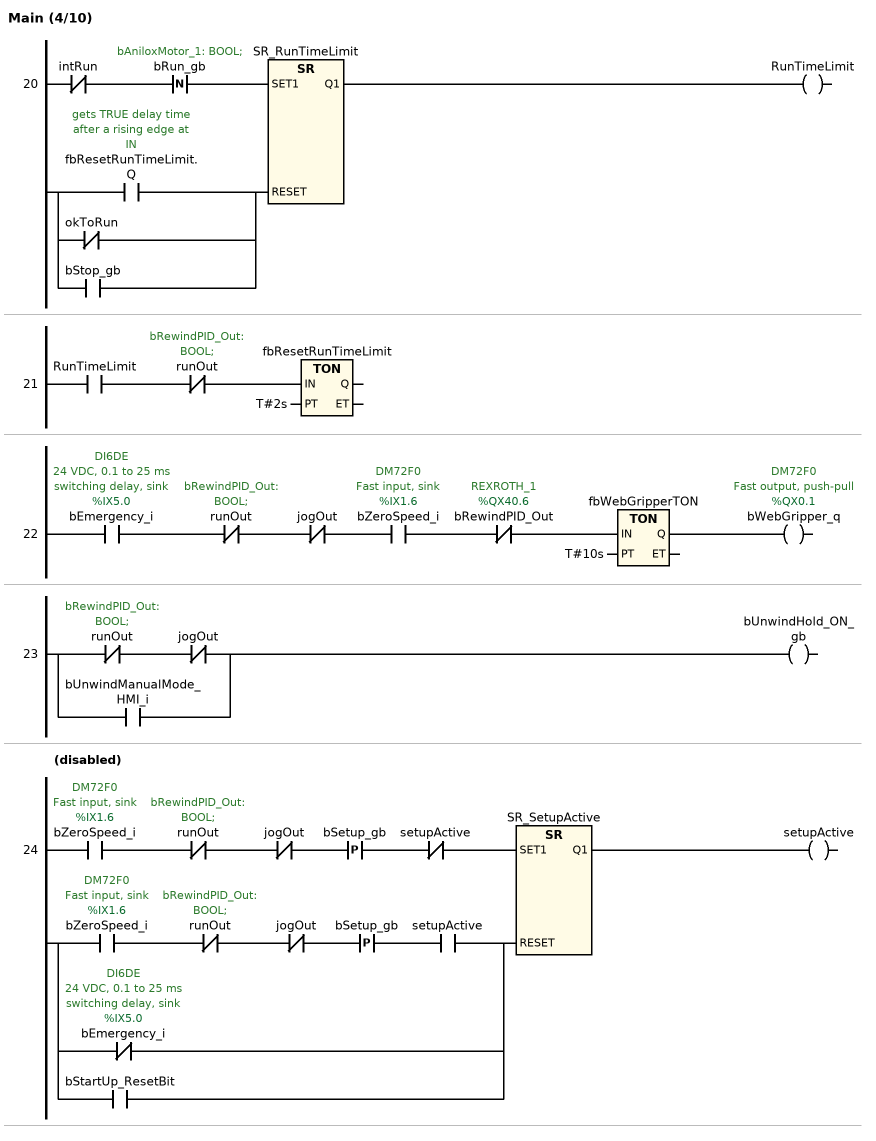
// NETWORK 20
//   bRun_gb: bAniloxMotor_1: BOOL;
//   fbResetRunTimeLimit.Q: gets TRUE delay time after a rising edge at IN
_ft2(CLK := bRun_gb);
SR_RunTimeLimit(SET1 := NOT intRun AND _ft2.Q, RESET := fbResetRunTimeLimit.Q OR NOT okToRun OR bStop_gb); // SR
RunTimeLimit := SR_RunTimeLimit.Q1;

// NETWORK 21
//   runOut: bRewindPID_Out:BOOL;
fbResetRunTimeLimit(IN := RunTimeLimit AND NOT runOut, PT := T#2s); // TON

// NETWORK 22
//   bEmergency_i: DI6DE 24 VDC, 0.1 to 25 ms switching delay, sink | AT %IX5.0
//   runOut: bRewindPID_Out:BOOL;
//   bZeroSpeed_i: DM72F0 Fast input, sink | AT %IX1.6
//   bRewindPID_Out: REXROTH_1 | AT %QX40.6
//   bWebGripper_q: DM72F0 Fast output, push-pull | AT %QX0.1
fbWebGripperTON(IN := bEmergency_i AND NOT runOut AND NOT jogOut AND bZeroSpeed_i AND NOT bRewindPID_Out, PT := T#10s); // TON
bWebGripper_q := fbWebGripperTON.Q;

// NETWORK 23
//   runOut: bRewindPID_Out:BOOL;
bUnwindHold_ON_gb := NOT runOut AND NOT jogOut OR bUnwindManualMode_HMI_i;

// NETWORK 24 (disabled)
//   bZeroSpeed_i: DM72F0 Fast input, sink | AT %IX1.6
//   runOut: bRewindPID_Out:BOOL;
//   bEmergency_i: DI6DE 24 VDC, 0.1 to 25 ms switching delay, sink | AT %IX5.0
// _rt4(CLK := bSetup_gb);
// _rt5(CLK := bSetup_gb);
// SR_SetupActive(SET1 := bZeroSpeed_i AND NOT runOut AND NOT jogOut AND _rt4.Q AND NOT setupActive, RESET := bZeroSpeed_i AND NOT runOut AND NOT jogOut AND _rt5.Q AND setupActive OR NOT bEmergency_i OR bStartUp_ResetBit); // SR
// setupActive := SR_SetupActive.Q1;

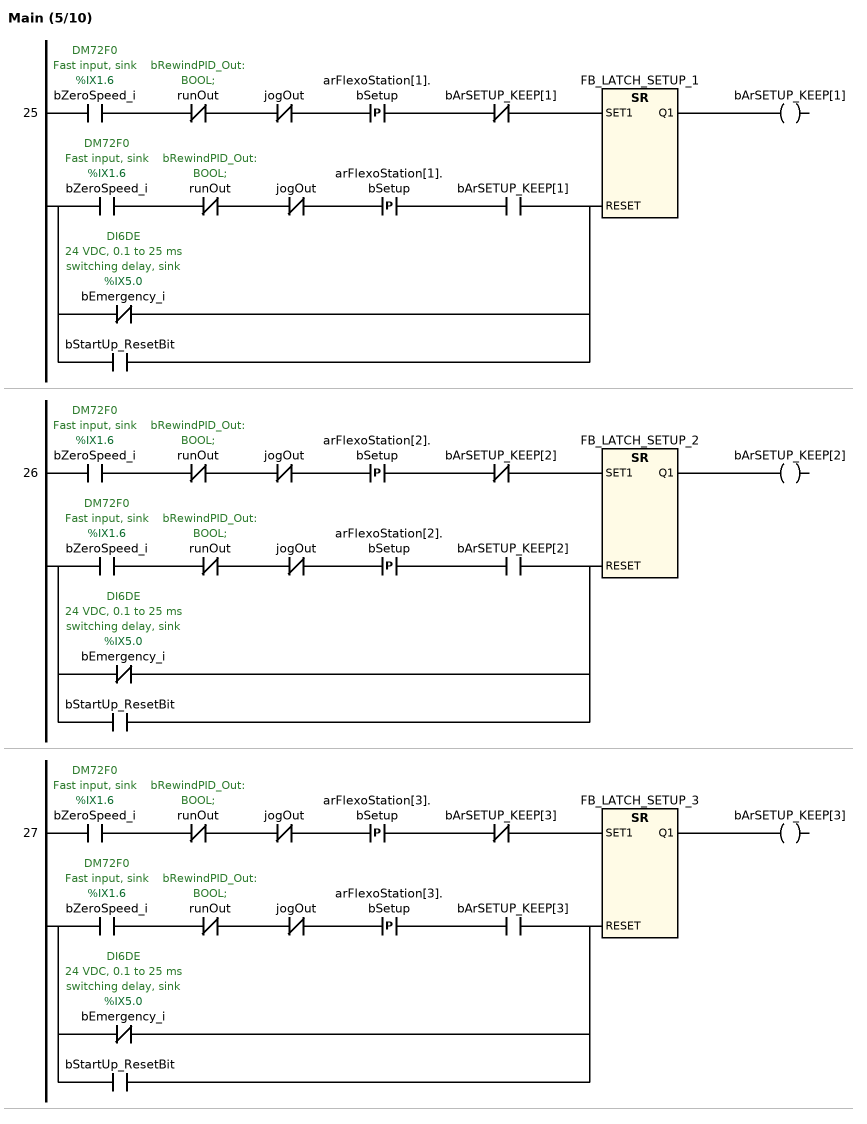
// NETWORK 25
//   bZeroSpeed_i: DM72F0 Fast input, sink | AT %IX1.6
//   runOut: bRewindPID_Out:BOOL;
//   bEmergency_i: DI6DE 24 VDC, 0.1 to 25 ms switching delay, sink | AT %IX5.0
_rt6(CLK := arFlexoStation[1].bSetup);
_rt7(CLK := arFlexoStation[1].bSetup);
FB_LATCH_SETUP_1(SET1 := bZeroSpeed_i AND NOT runOut AND NOT jogOut AND _rt6.Q AND NOT bArSETUP_KEEP[1], RESET := bZeroSpeed_i AND NOT runOut AND NOT jogOut AND _rt7.Q AND bArSETUP_KEEP[1] OR NOT bEmergency_i OR bStartUp_ResetBit); // SR
bArSETUP_KEEP[1] := FB_LATCH_SETUP_1.Q1;

// NETWORK 26
//   bZeroSpeed_i: DM72F0 Fast input, sink | AT %IX1.6
//   runOut: bRewindPID_Out:BOOL;
//   bEmergency_i: DI6DE 24 VDC, 0.1 to 25 ms switching delay, sink | AT %IX5.0
_rt8(CLK := arFlexoStation[2].bSetup);
_rt9(CLK := arFlexoStation[2].bSetup);
FB_LATCH_SETUP_2(SET1 := bZeroSpeed_i AND NOT runOut AND NOT jogOut AND _rt8.Q AND NOT bArSETUP_KEEP[2], RESET := bZeroSpeed_i AND NOT runOut AND NOT jogOut AND _rt9.Q AND bArSETUP_KEEP[2] OR NOT bEmergency_i OR bStartUp_ResetBit); // SR
bArSETUP_KEEP[2] := FB_LATCH_SETUP_2.Q1;

// NETWORK 27
//   bZeroSpeed_i: DM72F0 Fast input, sink | AT %IX1.6
//   runOut: bRewindPID_Out:BOOL;
//   bEmergency_i: DI6DE 24 VDC, 0.1 to 25 ms switching delay, sink | AT %IX5.0
_rt10(CLK := arFlexoStation[3].bSetup);
_rt11(CLK := arFlexoStation[3].bSetup);
FB_LATCH_SETUP_3(SET1 := bZeroSpeed_i AND NOT runOut AND NOT jogOut AND _rt10.Q AND NOT bArSETUP_KEEP[3], RESET := bZeroSpeed_i AND NOT runOut AND NOT jogOut AND _rt11.Q AND bArSETUP_KEEP[3] OR NOT bEmergency_i OR bStartUp_ResetBit); // SR
bArSETUP_KEEP[3] := FB_LATCH_SETUP_3.Q1;

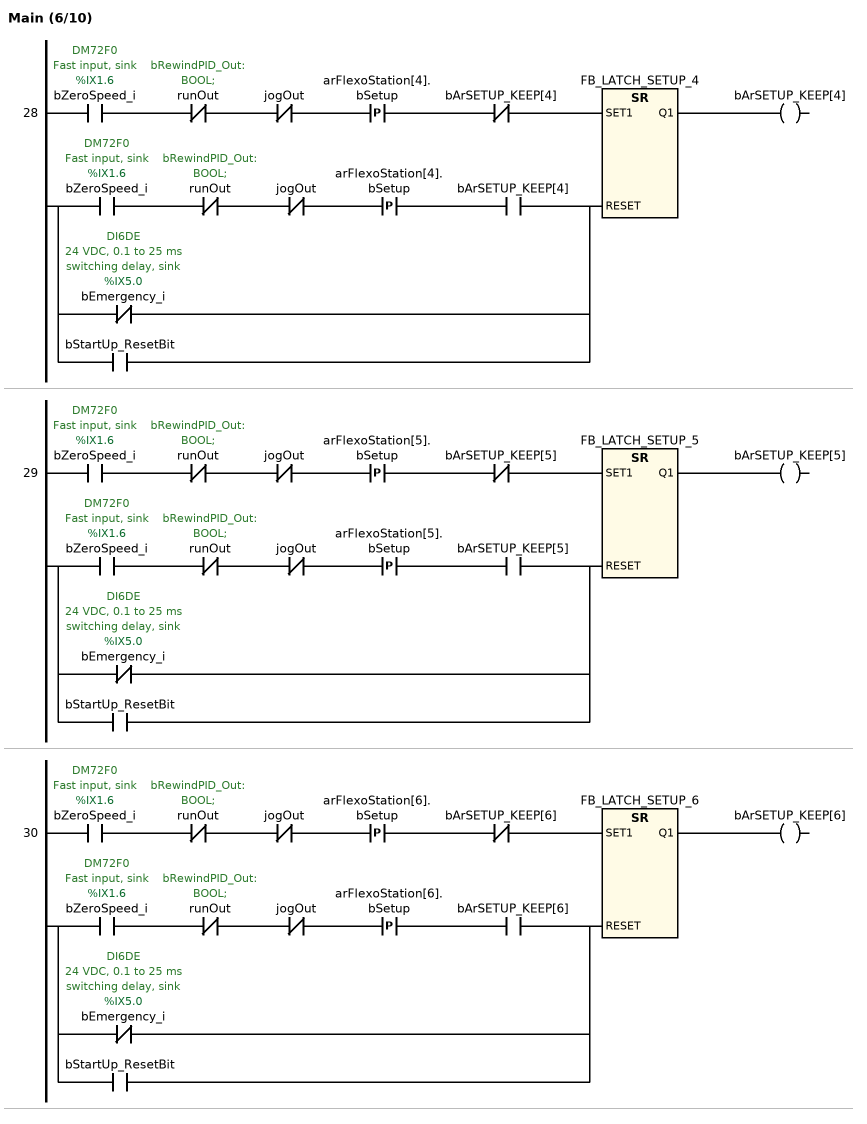
// NETWORK 28
//   bZeroSpeed_i: DM72F0 Fast input, sink | AT %IX1.6
//   runOut: bRewindPID_Out:BOOL;
//   bEmergency_i: DI6DE 24 VDC, 0.1 to 25 ms switching delay, sink | AT %IX5.0
_rt12(CLK := arFlexoStation[4].bSetup);
_rt13(CLK := arFlexoStation[4].bSetup);
FB_LATCH_SETUP_4(SET1 := bZeroSpeed_i AND NOT runOut AND NOT jogOut AND _rt12.Q AND NOT bArSETUP_KEEP[4], RESET := bZeroSpeed_i AND NOT runOut AND NOT jogOut AND _rt13.Q AND bArSETUP_KEEP[4] OR NOT bEmergency_i OR bStartUp_ResetBit); // SR
bArSETUP_KEEP[4] := FB_LATCH_SETUP_4.Q1;

// NETWORK 29
//   bZeroSpeed_i: DM72F0 Fast input, sink | AT %IX1.6
//   runOut: bRewindPID_Out:BOOL;
//   bEmergency_i: DI6DE 24 VDC, 0.1 to 25 ms switching delay, sink | AT %IX5.0
_rt14(CLK := arFlexoStation[5].bSetup);
_rt15(CLK := arFlexoStation[5].bSetup);
FB_LATCH_SETUP_5(SET1 := bZeroSpeed_i AND NOT runOut AND NOT jogOut AND _rt14.Q AND NOT bArSETUP_KEEP[5], RESET := bZeroSpeed_i AND NOT runOut AND NOT jogOut AND _rt15.Q AND bArSETUP_KEEP[5] OR NOT bEmergency_i OR bStartUp_ResetBit); // SR
bArSETUP_KEEP[5] := FB_LATCH_SETUP_5.Q1;

// NETWORK 30
//   bZeroSpeed_i: DM72F0 Fast input, sink | AT %IX1.6
//   runOut: bRewindPID_Out:BOOL;
//   bEmergency_i: DI6DE 24 VDC, 0.1 to 25 ms switching delay, sink | AT %IX5.0
_rt16(CLK := arFlexoStation[6].bSetup);
_rt17(CLK := arFlexoStation[6].bSetup);
FB_LATCH_SETUP_6(SET1 := bZeroSpeed_i AND NOT runOut AND NOT jogOut AND _rt16.Q AND NOT bArSETUP_KEEP[6], RESET := bZeroSpeed_i AND NOT runOut AND NOT jogOut AND _rt17.Q AND bArSETUP_KEEP[6] OR NOT bEmergency_i OR bStartUp_ResetBit); // SR
bArSETUP_KEEP[6] := FB_LATCH_SETUP_6.Q1;

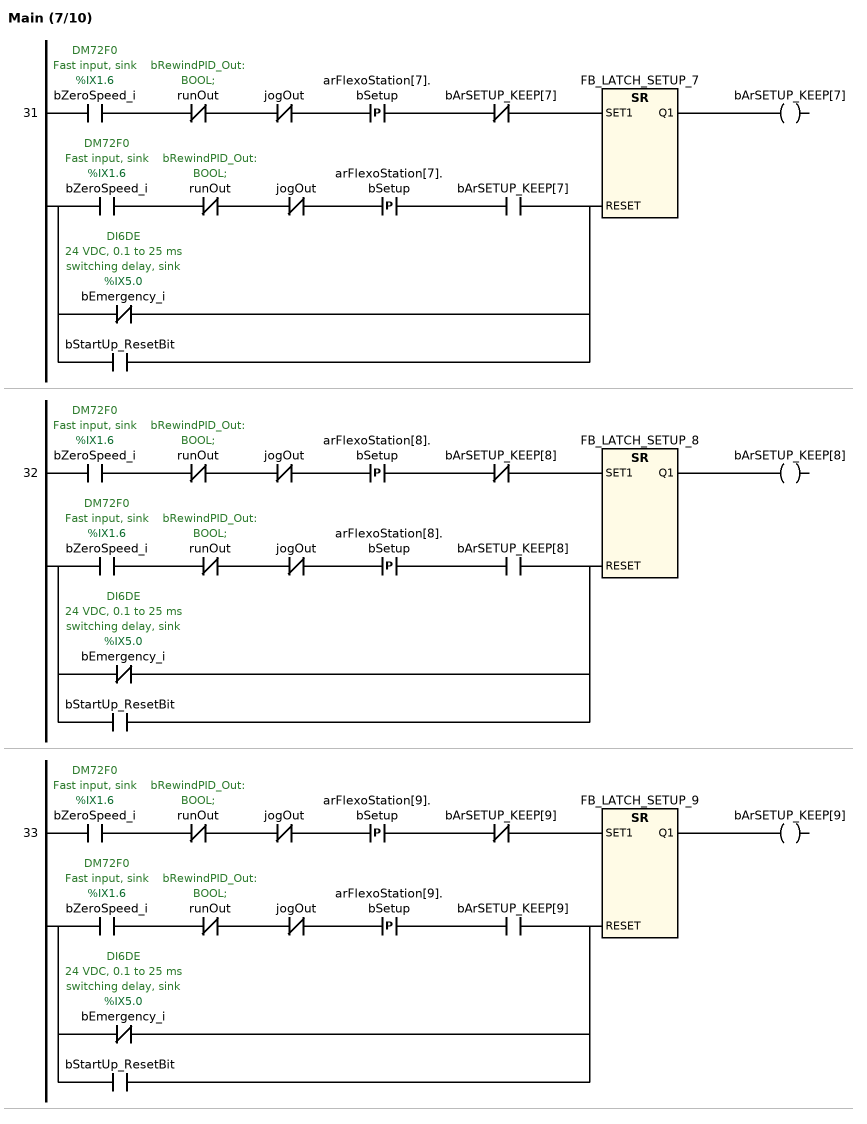
// NETWORK 31
//   bZeroSpeed_i: DM72F0 Fast input, sink | AT %IX1.6
//   runOut: bRewindPID_Out:BOOL;
//   bEmergency_i: DI6DE 24 VDC, 0.1 to 25 ms switching delay, sink | AT %IX5.0
_rt18(CLK := arFlexoStation[7].bSetup);
_rt19(CLK := arFlexoStation[7].bSetup);
FB_LATCH_SETUP_7(SET1 := bZeroSpeed_i AND NOT runOut AND NOT jogOut AND _rt18.Q AND NOT bArSETUP_KEEP[7], RESET := bZeroSpeed_i AND NOT runOut AND NOT jogOut AND _rt19.Q AND bArSETUP_KEEP[7] OR NOT bEmergency_i OR bStartUp_ResetBit); // SR
bArSETUP_KEEP[7] := FB_LATCH_SETUP_7.Q1;

// NETWORK 32
//   bZeroSpeed_i: DM72F0 Fast input, sink | AT %IX1.6
//   runOut: bRewindPID_Out:BOOL;
//   bEmergency_i: DI6DE 24 VDC, 0.1 to 25 ms switching delay, sink | AT %IX5.0
_rt20(CLK := arFlexoStation[8].bSetup);
_rt21(CLK := arFlexoStation[8].bSetup);
FB_LATCH_SETUP_8(SET1 := bZeroSpeed_i AND NOT runOut AND NOT jogOut AND _rt20.Q AND NOT bArSETUP_KEEP[8], RESET := bZeroSpeed_i AND NOT runOut AND NOT jogOut AND _rt21.Q AND bArSETUP_KEEP[8] OR NOT bEmergency_i OR bStartUp_ResetBit); // SR
bArSETUP_KEEP[8] := FB_LATCH_SETUP_8.Q1;

// NETWORK 33
//   bZeroSpeed_i: DM72F0 Fast input, sink | AT %IX1.6
//   runOut: bRewindPID_Out:BOOL;
//   bEmergency_i: DI6DE 24 VDC, 0.1 to 25 ms switching delay, sink | AT %IX5.0
_rt22(CLK := arFlexoStation[9].bSetup);
_rt23(CLK := arFlexoStation[9].bSetup);
FB_LATCH_SETUP_9(SET1 := bZeroSpeed_i AND NOT runOut AND NOT jogOut AND _rt22.Q AND NOT bArSETUP_KEEP[9], RESET := bZeroSpeed_i AND NOT runOut AND NOT jogOut AND _rt23.Q AND bArSETUP_KEEP[9] OR NOT bEmergency_i OR bStartUp_ResetBit); // SR
bArSETUP_KEEP[9] := FB_LATCH_SETUP_9.Q1;

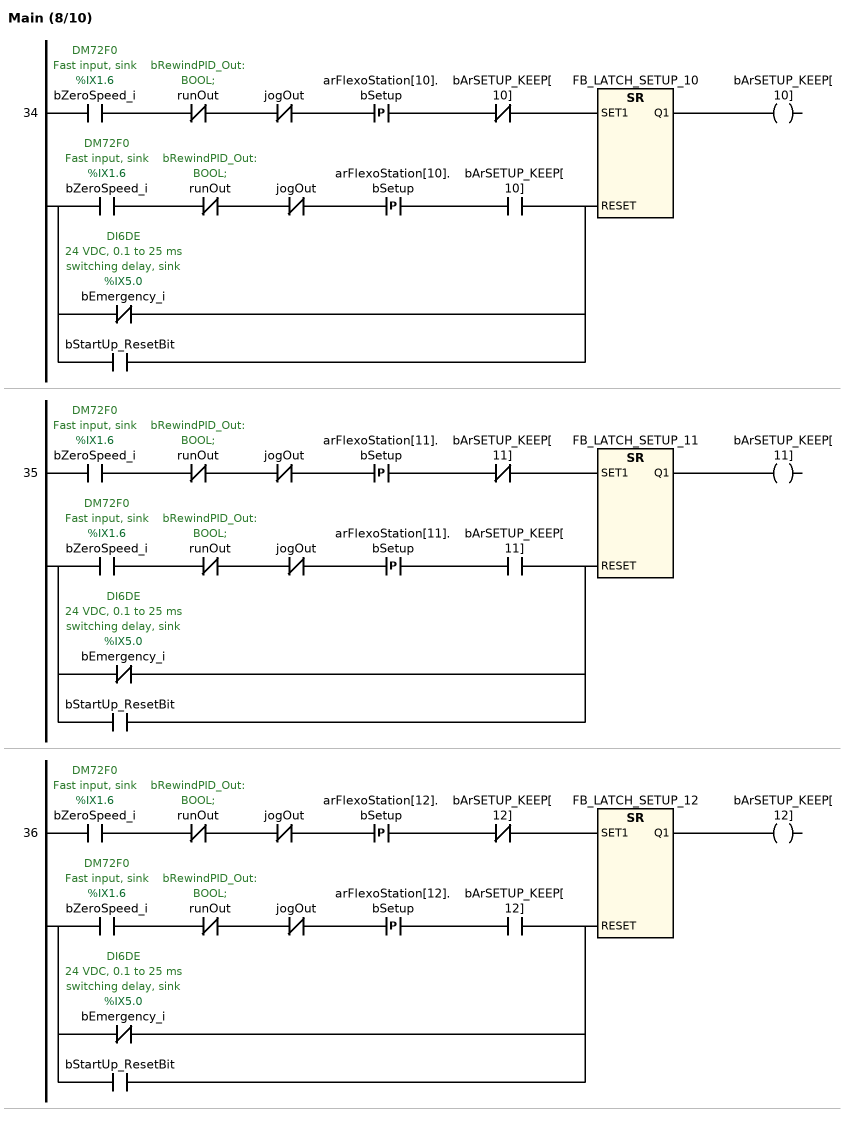
// NETWORK 34
//   bZeroSpeed_i: DM72F0 Fast input, sink | AT %IX1.6
//   runOut: bRewindPID_Out:BOOL;
//   bEmergency_i: DI6DE 24 VDC, 0.1 to 25 ms switching delay, sink | AT %IX5.0
_rt24(CLK := arFlexoStation[10].bSetup);
_rt25(CLK := arFlexoStation[10].bSetup);
FB_LATCH_SETUP_10(SET1 := bZeroSpeed_i AND NOT runOut AND NOT jogOut AND _rt24.Q AND NOT bArSETUP_KEEP[10], RESET := bZeroSpeed_i AND NOT runOut AND NOT jogOut AND _rt25.Q AND bArSETUP_KEEP[10] OR NOT bEmergency_i OR bStartUp_ResetBit); // SR
bArSETUP_KEEP[10] := FB_LATCH_SETUP_10.Q1;

// NETWORK 35
//   bZeroSpeed_i: DM72F0 Fast input, sink | AT %IX1.6
//   runOut: bRewindPID_Out:BOOL;
//   bEmergency_i: DI6DE 24 VDC, 0.1 to 25 ms switching delay, sink | AT %IX5.0
_rt26(CLK := arFlexoStation[11].bSetup);
_rt27(CLK := arFlexoStation[11].bSetup);
FB_LATCH_SETUP_11(SET1 := bZeroSpeed_i AND NOT runOut AND NOT jogOut AND _rt26.Q AND NOT bArSETUP_KEEP[11], RESET := bZeroSpeed_i AND NOT runOut AND NOT jogOut AND _rt27.Q AND bArSETUP_KEEP[11] OR NOT bEmergency_i OR bStartUp_ResetBit); // SR
bArSETUP_KEEP[11] := FB_LATCH_SETUP_11.Q1;

// NETWORK 36
//   bZeroSpeed_i: DM72F0 Fast input, sink | AT %IX1.6
//   runOut: bRewindPID_Out:BOOL;
//   bEmergency_i: DI6DE 24 VDC, 0.1 to 25 ms switching delay, sink | AT %IX5.0
_rt28(CLK := arFlexoStation[12].bSetup);
_rt29(CLK := arFlexoStation[12].bSetup);
FB_LATCH_SETUP_12(SET1 := bZeroSpeed_i AND NOT runOut AND NOT jogOut AND _rt28.Q AND NOT bArSETUP_KEEP[12], RESET := bZeroSpeed_i AND NOT runOut AND NOT jogOut AND _rt29.Q AND bArSETUP_KEEP[12] OR NOT bEmergency_i OR bStartUp_ResetBit); // SR
bArSETUP_KEEP[12] := FB_LATCH_SETUP_12.Q1;

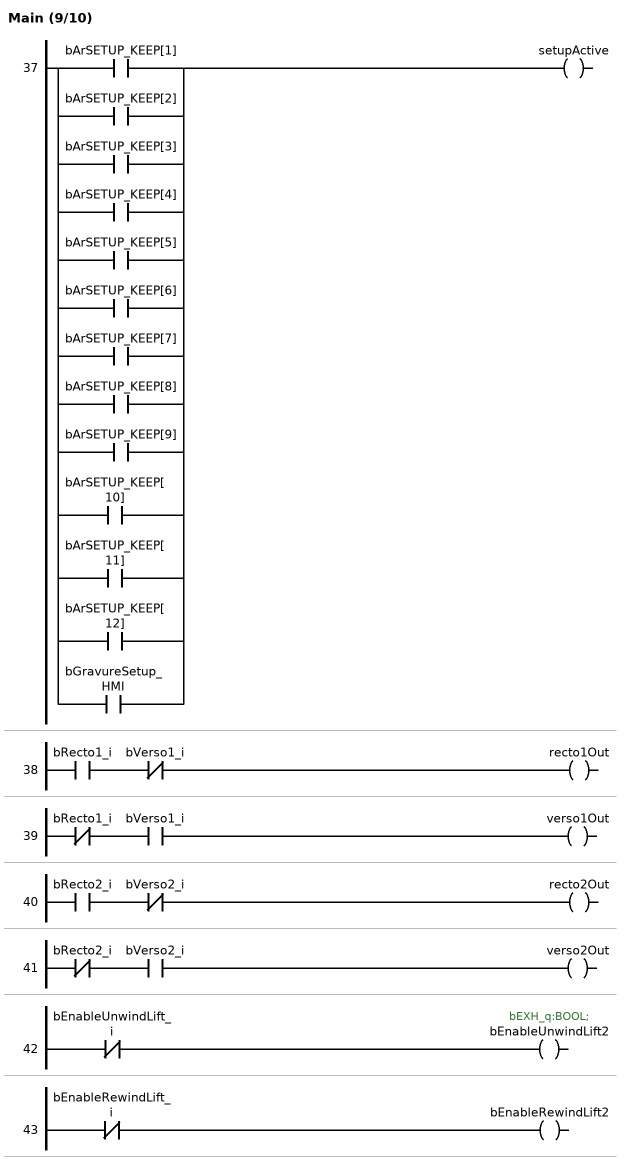
// NETWORK 37
setupActive := bArSETUP_KEEP[1] OR bArSETUP_KEEP[2] OR bArSETUP_KEEP[3] OR bArSETUP_KEEP[4] OR bArSETUP_KEEP[5] OR bArSETUP_KEEP[6] OR bArSETUP_KEEP[7] OR bArSETUP_KEEP[8] OR bArSETUP_KEEP[9] OR bArSETUP_KEEP[10] OR bArSETUP_KEEP[11] OR bArSETUP_KEEP[12] OR bGravureSetup_HMI;

// NETWORK 38
recto1Out := bRecto1_i AND NOT bVerso1_i;

// NETWORK 39
verso1Out := NOT bRecto1_i AND bVerso1_i;

// NETWORK 40
recto2Out := bRecto2_i AND NOT bVerso2_i;

// NETWORK 41
verso2Out := NOT bRecto2_i AND bVerso2_i;

// NETWORK 42
//   bEnableUnwindLift2: bEXH_q:BOOL;
bEnableUnwindLift2 := NOT bEnableUnwindLift_i;

// NETWORK 43
bEnableRewindLift2 := NOT bEnableRewindLift_i;

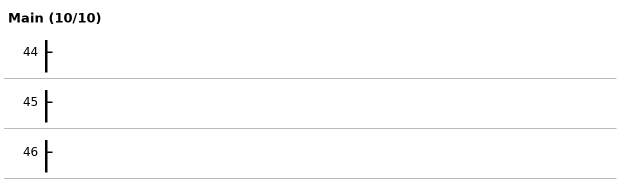
// NETWORK 44

// NETWORK 45

// NETWORK 46

END_PROGRAM

// MyController/Application/COUNTER/COUNTER
PROGRAM COUNTER
VAR

DESIRED_COUNT:DINT;
	
COUNT_RESET:BOOL;
COUNTER_ON:BOOL;


BEGIN_COUNT:DINT;

ACTUAL_COUNT:DINT;

//COUNT_TOT_RESET:BOOL;
//COUNTER_TOT_ON:BOOL;
TOT_COUNTER_ON:BOOL;
TOT_RESET_ON:BOOL;

BEGIN_TOT_COUNT:DINT;
BASE_TOT_FINAL_CNT:DINT;
ACTUAL_TOT_COUNT:DINT;

TOT_COUNT_RESET:BOOL;


	rInchActualCountPPR: REAL;
	
	
	rInchActualTotCountPPR: REAL;
	rInchActualTotCount:REAL;
	
	rRepeatLimited:REAL; (*IN INCHES*)
	rLineShaftGBXLimited:REAL;
END_VAR

	(*REPEAT*)
	IF rRepeat_HMI_i = 0.0 THEN
		rRepeat_HMI_i := 1.0;
		rRepeatLimited	:= 1.0;
	ELSE rRepeatLimited	:= rRepeat_HMI_i;
	END_IF
	(*GEARBOX*)
	IF rLineShaftGBX_HMI_i = 0.0 THEN
		rLineShaftGBX_HMI_i 	:= 1.0;  //rLineShaftGBX_HMI_i
		rLineShaftGBXLimited	:= 1.0;
	ELSE rLineShaftGBXLimited := rLineShaftGBX_HMI_i;
	END_IF
	

	rRepeatCount_HMI_q :=  rInchActualCount/rRepeatLimited;

	(*COUNTER*)
	IF bResetCount_HMI_i = 1  THEN
		BEGIN_COUNT := BASE_FINAL_CNT;	//THATS WHERE WE START COUNTING
		ACTUAL_COUNT := 0;
		COUNT_RESET := 0;
	END_IF
	IF BASE_FINAL_CNT >= BEGIN_COUNT AND bCounterOn_HMI_i = 1  THEN
		ACTUAL_COUNT	:=	BASE_FINAL_CNT - BEGIN_COUNT;
	ELSIF COUNTER_ON = 0  THEN
		BEGIN_COUNT	:=	BASE_FINAL_CNT - ACTUAL_COUNT;
	END_IF
	rInchActualCountPPR := (GVL_ENCODER.rInchPerTurn * ACTUAL_COUNT)/(rLineShaftGBXLimited);
	rInchActualCount	:= rInchActualCountPPR/4096;
	rRepeatCount_HMI_q :=  ((ACTUAL_COUNT/1024)*uiCOUNT_BASE)/1000;//rInchActualCount/rRepeatLimited;


	
	(*TOTALIZER*)
	IF bTotResetCount_HMI_i = 1  THEN
		BEGIN_TOT_COUNT := BASE_FINAL_CNT;	//THATS WHERE WE START COUNTING
		ACTUAL_TOT_COUNT := 0;
	END_IF
	IF BASE_FINAL_CNT >= BEGIN_TOT_COUNT AND bTotCounterOn_HMI_i = 1  THEN
		ACTUAL_TOT_COUNT	:=	BASE_FINAL_CNT - BEGIN_TOT_COUNT;
	ELSIF TOT_COUNTER_ON = 0  THEN
		BEGIN_TOT_COUNT	:=	BASE_FINAL_CNT - ACTUAL_TOT_COUNT;
	END_IF
	rInchActualTotCountPPR := (GVL_ENCODER.rInchPerTurn * ACTUAL_TOT_COUNT)/(rLineShaftGBXLimited);
	rInchActualTotCount	:= rInchActualTotCountPPR/4096;
	rRepeatTotCount_HMI_q :=  ((ACTUAL_TOT_COUNT/1024)*uiCOUNT_BASE)/10000;//rInchActualTotCount/rRepeatLimited;

	
	(*COUNT REACHED*)
	IF rRepeatCount_HMI_q <= rDesiredCount_HMI_i THEN
		GVL_GENERAL.COUNTER_REACHED := 1;
	ELSE
		GVL_GENERAL.COUNTER_REACHED := 0;
	END_IF

END_PROGRAM

// MyController/Application/OPTIONS/AccessCode
PROGRAM AccessCode
VAR


END_VAR


	IF uiAccessCode = 2032 THEN
		bAccessGranted := TRUE;
	ELSE
		bAccessGranted := FALSE;
	END_IF

END_PROGRAM

// MyController/Application/CAN_NETWORK
PROGRAM CAN_NETWORK
VAR
	NewVal1 :UINT := 5;
	NewVal2 :UINT := 5;
	Result :UINT := 0;
	

	
	bVar1:BOOL:=FALSE;
	bVar2:BOOL:=FALSE;
	bVar3:BOOL:=FALSE;
	bVar4:BOOL:=FALSE;
	bVar5:BOOL:=FALSE;
	bVar6:BOOL:=FALSE;
	bVar7:BOOL:=FALSE;
	bVar8:BOOL:=FALSE;
	
	bVar9:BOOL:=FALSE;
	bVar10:BOOL:=FALSE;
	bVar11:BOOL:=FALSE;
	bVar12:BOOL:=FALSE;
	
	
	
	byTEST:BYTE;
	
	wStationBrd1_UpperByte:WORD;
	wStationBrd1_LowerByte:WORD;
	
	wStationBrd2_UpperByte:WORD;
	wStationBrd2_LowerByte:WORD;
	
	wStationBrd3_UpperByte:WORD;
	wStationBrd3_LowerByte:WORD;
	
	wStationBrd4_UpperByte:WORD;
	wStationBrd4_LowerByte:WORD;
	
	wStationBrd5_UpperByte:WORD;
	wStationBrd5_LowerByte:WORD;
	
	wStationBrd6_UpperByte:WORD;
	wStationBrd6_LowerByte:WORD;
	
	wStationBrd7_UpperByte:WORD;
	wStationBrd7_LowerByte:WORD;
	
	wStationBrd8_UpperByte:WORD;
	wStationBrd8_LowerByte:WORD;
	
	wStationBrd9_UpperByte:WORD;
	wStationBrd9_LowerByte:WORD;
	
	wStationBrd10_UpperByte:WORD;
	wStationBrd10_LowerByte:WORD;
	
	wStationBrd11_UpperByte:WORD;
	wStationBrd11_LowerByte:WORD;
	
	wStationBrd12_UpperByte:WORD;
	wStationBrd12_LowerByte:WORD;
	
	fbRUNout: TP;
	bBogus3 :BYTE;
	bBogus1: BYTE;
	bBogus2: BYTE;
	bBogus4: BYTE;
	bBogus5: BYTE;
	bAniloxKickoff6_q: BOOL;
	bAniloxKickoff7_q: BOOL;
	bAniloxKickoff8_q: BOOL;
	bAniloxKickoff9_q: BOOL;
	bAniloxKickoff10_q: BOOL;

	i: INT;
	
	wStationBrd_UpperByte:	ARRAY[1..20]OF WORD;
	wStationBrd_LowerByte:	ARRAY[1..20]OF WORD;
	
	
	wRelayBrd_UpperByte:	ARRAY[1..20]OF WORD;
	wRelayBrd_LowerByte:	ARRAY[1..20]OF WORD;
	
	bRegAdvanceRelay_q:BOOL;
	bRegRetardRelay_q:BOOL;
	
	
	
	bSpareRelay:BOOL:=FALSE;
	bAniloxRelay:BOOL:=FALSE;

	bPlateKickOff:BOOL:=FALSE;
	bAniloxKickOff:BOOL:=FALSE;

	
	bComHeart_StationBoard:	ARRAY[1..20]OF BOOL;
	bComHeart_RelayBoard:	ARRAY[1..20]OF BOOL;
	bComHeartBeat_Bypass_CAN_i: ARRAY[1..20]OF BOOL;
	
	
	
	TEST_ON: TON;
END_VAR


//wStationBrd4_gb	:=	uiStationBrd4_gb;
//wStationBrd1_gb:WORD;
//wStationBrd2_gb:WORD;
//wStationBrd3_gb:WORD;
//wStationBrd4_gb:WORD;


FOR i:=1 TO 20 BY 1 DO

	wStationBrd_UpperByte[i] 	:= SHL(BYTE_TO_WORD(PACK(bGreenLightRunStatus_q,(NOT readyInd),bArAniloxMotor_KEEP[i],bArAniloxKickoff_KEEP[i],FALSE,FALSE,FALSE,FALSE)),8);
	wStationBrd_LowerByte[i] 	:= BYTE_TO_WORD(PACK(bArPlateKickoff_KEEP[i],bArIR_KEEP[i],bArSETUP_KEEP[i],bInkingOn_KEEP,bPrintingOn_KEEP,arFlexoStation[i].bSpare1_q,arFlexoStation[i].bSpare2_q,arFlexoStation[i].bSpare3_q));
	wStationBrd_LED_q[i] 		:= WORD_TO_UINT(wStationBrd_UpperByte[i] OR wStationBrd_LowerByte[i]);

END_FOR

bIncSpeed_q	:=	bEmergency_i	AND (arFlexoStation[1].bRunPlus OR arFlexoStation[2].bRunPlus OR arFlexoStation[3].bRunPlus OR arFlexoStation[4].bRunPlus	OR
								arFlexoStation[5].bRunPlus OR arFlexoStation[6].bRunPlus OR arFlexoStation[7].bRunPlus OR arFlexoStation[8].bRunPlus	OR
								arFlexoStation[9].bRunPlus OR arFlexoStation[10].bRunPlus OR arFlexoStation[11].bRunPlus OR arFlexoStation[12].bRunPlus OR arFlexoStation[13].bRunPlus) AND fbRUNOUT_REAL.Q;
			
bDecSpeed_q	:=	bEmergency_i	AND (arFlexoStation[1].bRunMinus OR arFlexoStation[2].bRunMinus OR arFlexoStation[3].bRunMinus OR arFlexoStation[4].bRunMinus	OR
								arFlexoStation[5].bRunMinus OR arFlexoStation[6].bRunMinus OR arFlexoStation[7].bRunMinus OR arFlexoStation[8].bRunMinus	OR
								arFlexoStation[9].bRunMinus OR arFlexoStation[10].bRunMinus OR arFlexoStation[11].bRunMinus OR arFlexoStation[12].bRunMinus OR arFlexoStation[13].bRunMinus) AND fbRUNOUT_REAL.Q;




	
ArFlexoStation[1].bRegAdvance_q	:=	(ArFlexoStation[1].bRegAdvance OR bRegAdvance_1_HMI) AND (NOT ArFlexoStation[1].bRegRetard_q);
ArFlexoStation[1].bRegRetard_q	:= 	(ArFlexoStation[1].bRegRetard OR  bRegRetard_1_HMI) AND (NOT ArFlexoStation[1].bRegAdvance_q);

ArFlexoStation[2].bRegAdvance_q	:=	(ArFlexoStation[2].bRegAdvance OR bRegAdvance_2_HMI) AND (NOT ArFlexoStation[2].bRegRetard_q);
ArFlexoStation[2].bRegRetard_q	:= 	(ArFlexoStation[2].bRegRetard OR  bRegRetard_2_HMI) AND (NOT ArFlexoStation[2].bRegAdvance_q);

ArFlexoStation[3].bRegAdvance_q	:=	(ArFlexoStation[3].bRegAdvance OR bRegAdvance_3_HMI) AND (NOT ArFlexoStation[3].bRegRetard_q);
ArFlexoStation[3].bRegRetard_q	:= 	(ArFlexoStation[3].bRegRetard OR  bRegRetard_3_HMI) AND (NOT ArFlexoStation[3].bRegAdvance_q);

ArFlexoStation[5].bRegAdvance_q	:=	(ArFlexoStation[4].bRegAdvance OR bRegAdvance_4_HMI) AND (NOT ArFlexoStation[4].bRegRetard_q);
ArFlexoStation[5].bRegRetard_q	:= 	(ArFlexoStation[4].bRegRetard OR  bRegRetard_4_HMI) AND (NOT ArFlexoStation[4].bRegAdvance_q);

ArFlexoStation[6].bRegAdvance_q	:=	(ArFlexoStation[5].bRegAdvance OR bRegAdvance_5_HMI) AND (NOT ArFlexoStation[5].bRegRetard_q);
ArFlexoStation[6].bRegRetard_q	:= 	(ArFlexoStation[5].bRegRetard OR  bRegRetard_5_HMI) AND (NOT ArFlexoStation[5].bRegAdvance_q);

ArFlexoStation[7].bRegAdvance_q	:=	(ArFlexoStation[6].bRegAdvance OR bRegAdvance_6_HMI) AND (NOT ArFlexoStation[6].bRegRetard_q);
ArFlexoStation[7].bRegRetard_q	:= 	(ArFlexoStation[6].bRegRetard OR  bRegRetard_6_HMI) AND (NOT ArFlexoStation[6].bRegAdvance_q);

ArFlexoStation[9].bRegAdvance_q	:=	(ArFlexoStation[7].bRegAdvance OR bRegAdvance_7_HMI) AND (NOT ArFlexoStation[7].bRegRetard_q);
ArFlexoStation[9].bRegRetard_q	:= 	(ArFlexoStation[7].bRegRetard OR  bRegRetard_7_HMI) AND (NOT ArFlexoStation[7].bRegAdvance_q);

ArFlexoStation[10].bRegAdvance_q	:=	(ArFlexoStation[8].bRegAdvance OR bRegAdvance_8_HMI) AND (NOT ArFlexoStation[8].bRegRetard_q);
ArFlexoStation[10].bRegRetard_q	:= 	(ArFlexoStation[8].bRegRetard OR  bRegRetard_8_HMI) AND (NOT ArFlexoStation[8].bRegAdvance_q);


ArFlexoStation[11].bRegAdvance_q	:=	(ArFlexoStation[9].bRegAdvance OR bRegAdvance_9_HMI) AND (NOT ArFlexoStation[9].bRegRetard_q);
ArFlexoStation[11].bRegRetard_q	:= 	(ArFlexoStation[9].bRegRetard OR  bRegRetard_9_HMI) AND (NOT ArFlexoStation[9].bRegAdvance_q);

	
ArFlexoStation[12].bRegAdvance_q	:=	(ArFlexoStation[10].bRegAdvance OR bRegAdvance_10_HMI) AND (NOT ArFlexoStation[10].bRegRetard_q);
ArFlexoStation[12].bRegRetard_q		:= 	(ArFlexoStation[10].bRegRetard OR  bRegRetard_10_HMI) AND (NOT ArFlexoStation[10].bRegAdvance_q);

ArFlexoStation[13].bRegAdvance_q	:=	(ArFlexoStation[11].bRegAdvance OR bRegAdvance_11_HMI) AND (NOT ArFlexoStation[11].bRegRetard_q);
ArFlexoStation[13].bRegRetard_q		:= 	(ArFlexoStation[11].bRegRetard OR  bRegRetard_11_HMI) AND (NOT ArFlexoStation[11].bRegAdvance_q);
	
ArFlexoStation[14].bRegAdvance_q	:=	(ArFlexoStation[12].bRegAdvance OR bRegAdvance_12_HMI) AND (NOT ArFlexoStation[12].bRegRetard_q);
ArFlexoStation[14].bRegRetard_q		:= 	(ArFlexoStation[12].bRegRetard OR  bRegRetard_12_HMI) AND (NOT ArFlexoStation[12].bRegAdvance_q);



//*****************************************************************
//THIS PART DECODES THE SIGNAL GIVEN BY CORRESPONDING STATION BOARD	
//wStationBrd1_gb : h7F;
//*****************************************************************
	//bAniloxMtr_1	:= TRUE;
	//bAniloxKickOff_1	:= FALSE;
				
	//bPlateKickoff_1	:= FALSE;
	//			bInfraRed_1		:= FALSE;
	//			bRegAdvance_1	:= FALSE;
	//			bRegRetard_1		:= FALSE;
	//			bRunPlus_1		:= FALSE;
	//			bRunMinus_1		:= FALSE;
	//			bJog_1			:= FALSE;
	//			bStop_1			:= FALSE;
	//			GVL_KEY.bSetup_1	:= FALSE;
	//			GVL_KEY.bInkingOn_1	:= FALSE;
	//			GVL_KEY.bPrintingOn_1 := FALSE;


//wArStationBrd[1] ;	//:= UINT_TO_WORD(uiStationBrd1_gb);
i:=1;

FOR i:=1 TO 20 BY 1 DO


	CASE	wArStationBrd[i]	OF
	
	16#7D:	//ANILOX MOTOR
	
				arFlexoStation[i].bAniloxMtr 			:= TRUE;
				arFlexoStation[i].bAniloxKickOff 		:= FALSE;
				arFlexoStation[i].bPlateKickoff 		:= FALSE;
				arFlexoStation[i].bInfraRed 			:= FALSE;
				arFlexoStation[i].bRegAdvance			:= FALSE;
				arFlexoStation[i].bRegRetard			:= FALSE;
				arFlexoStation[i].bRunPlus				:= FALSE;
				arFlexoStation[i].bRunMinus				:= FALSE;
				arFlexoStation[i].bJog					:= FALSE;
				arFlexoStation[i].bStop					:= FALSE;
				arFlexoStation[i].bSetup				:= FALSE;
				arFlexoStation[i].bInkingOn				:= FALSE;
				arFlexoStation[i].bPrintingOn			:= FALSE;
				
				
				
	16#BD:	//ANILOX KICKOFF

				arFlexoStation[i].bAniloxMtr 			:= FALSE;
				arFlexoStation[i].bAniloxKickOff 		:= TRUE;
				arFlexoStation[i].bPlateKickoff 		:= FALSE;
				arFlexoStation[i].bInfraRed 			:= FALSE;
				arFlexoStation[i].bRegAdvance			:= FALSE;
				arFlexoStation[i].bRegRetard			:= FALSE;
				arFlexoStation[i].bRunPlus				:= FALSE;
				arFlexoStation[i].bRunMinus				:= FALSE;
				arFlexoStation[i].bJog					:= FALSE;
				arFlexoStation[i].bStop					:= FALSE;
				arFlexoStation[i].bSetup				:= FALSE;
				arFlexoStation[i].bInkingOn				:= FALSE;
				arFlexoStation[i].bPrintingOn			:= FALSE;
				
	16#DD:	//PLATE KICKOFF

				arFlexoStation[i].bAniloxMtr 			:= FALSE;
				arFlexoStation[i].bAniloxKickOff 		:= FALSE;
				arFlexoStation[i].bPlateKickoff 		:= TRUE;
				arFlexoStation[i].bInfraRed 			:= FALSE;
				arFlexoStation[i].bRegAdvance			:= FALSE;
				arFlexoStation[i].bRegRetard			:= FALSE;
				arFlexoStation[i].bRunPlus				:= FALSE;
				arFlexoStation[i].bRunMinus				:= FALSE;
				arFlexoStation[i].bJog					:= FALSE;
				arFlexoStation[i].bStop					:= FALSE;
				arFlexoStation[i].bSetup				:= FALSE;
				arFlexoStation[i].bInkingOn				:= FALSE;
				arFlexoStation[i].bPrintingOn			:= FALSE;
				
	16#ED:	//IR

				arFlexoStation[i].bAniloxMtr 			:= FALSE;
				arFlexoStation[i].bAniloxKickOff 		:= FALSE;
				arFlexoStation[i].bPlateKickoff 		:= FALSE;
				arFlexoStation[i].bInfraRed 			:= TRUE;
				arFlexoStation[i].bRegAdvance			:= FALSE;
				arFlexoStation[i].bRegRetard			:= FALSE;
				arFlexoStation[i].bRunPlus				:= FALSE;
				arFlexoStation[i].bRunMinus				:= FALSE;
				arFlexoStation[i].bJog					:= FALSE;
				arFlexoStation[i].bStop					:= FALSE;
				arFlexoStation[i].bSetup				:= FALSE;
				arFlexoStation[i].bInkingOn				:= FALSE;
				arFlexoStation[i].bPrintingOn			:= FALSE;
	
	16#BB:	//SETUP

				arFlexoStation[i].bAniloxMtr 			:= FALSE;
				arFlexoStation[i].bAniloxKickOff 		:= FALSE;
				arFlexoStation[i].bPlateKickoff 		:= FALSE;
				arFlexoStation[i].bInfraRed 			:= FALSE;
				arFlexoStation[i].bRegAdvance			:= FALSE;
				arFlexoStation[i].bRegRetard			:= FALSE;
				arFlexoStation[i].bRunPlus				:= FALSE;
				arFlexoStation[i].bRunMinus				:= FALSE;
				arFlexoStation[i].bJog					:= FALSE;
				arFlexoStation[i].bStop					:= FALSE;
				arFlexoStation[i].bSetup				:= TRUE;
				arFlexoStation[i].bInkingOn				:= FALSE;
				arFlexoStation[i].bPrintingOn			:= FALSE;
	
	16#DB:	//INKING ON

				arFlexoStation[i].bAniloxMtr 			:= FALSE;
				arFlexoStation[i].bAniloxKickOff 		:= FALSE;
				arFlexoStation[i].bPlateKickoff 		:= FALSE;
				arFlexoStation[i].bInfraRed 			:= FALSE;
				arFlexoStation[i].bRegAdvance			:= FALSE;
				arFlexoStation[i].bRegRetard			:= FALSE;
				arFlexoStation[i].bRunPlus				:= FALSE;
				arFlexoStation[i].bRunMinus				:= FALSE;
				arFlexoStation[i].bJog					:= FALSE;
				arFlexoStation[i].bStop					:= FALSE;
				arFlexoStation[i].bSetup				:= FALSE;
				arFlexoStation[i].bInkingOn				:= TRUE;
				arFlexoStation[i].bPrintingOn			:= FALSE;
	
		
	
	16#EB:	//PRINTING ON

				arFlexoStation[i].bAniloxMtr 			:= FALSE;
				arFlexoStation[i].bAniloxKickOff 		:= FALSE;
				arFlexoStation[i].bPlateKickoff 		:= FALSE;
				arFlexoStation[i].bInfraRed 			:= FALSE;
				arFlexoStation[i].bRegAdvance			:= FALSE;
				arFlexoStation[i].bRegRetard			:= FALSE;
				arFlexoStation[i].bRunPlus				:= FALSE;
				arFlexoStation[i].bRunMinus				:= FALSE;
				arFlexoStation[i].bJog					:= FALSE;
				arFlexoStation[i].bStop					:= FALSE;
				arFlexoStation[i].bSetup				:= FALSE;
				arFlexoStation[i].bInkingOn				:= FALSE;
				arFlexoStation[i].bPrintingOn			:= TRUE;
				
	16#BE:	//REG ADVANCE

				arFlexoStation[i].bAniloxMtr 			:= FALSE;
				arFlexoStation[i].bAniloxKickOff 		:= FALSE;
				arFlexoStation[i].bPlateKickoff 		:= FALSE;
				arFlexoStation[i].bInfraRed 			:= FALSE;
				arFlexoStation[i].bRegAdvance			:= TRUE;
				arFlexoStation[i].bRegRetard			:= FALSE;
				arFlexoStation[i].bRunPlus				:= FALSE;
				arFlexoStation[i].bRunMinus				:= FALSE;
				arFlexoStation[i].bJog					:= FALSE;
				arFlexoStation[i].bStop					:= FALSE;
				arFlexoStation[i].bSetup				:= FALSE;
				arFlexoStation[i].bInkingOn				:= FALSE;
				arFlexoStation[i].bPrintingOn			:= FALSE;


16#7E:	//REG RETARD

				arFlexoStation[i].bAniloxMtr 			:= FALSE;
				arFlexoStation[i].bAniloxKickOff 		:= FALSE;
				arFlexoStation[i].bPlateKickoff 		:= FALSE;
				arFlexoStation[i].bInfraRed 			:= FALSE;
				arFlexoStation[i].bRegAdvance			:= FALSE;
				arFlexoStation[i].bRegRetard			:= TRUE;
				arFlexoStation[i].bRunPlus				:= FALSE;
				arFlexoStation[i].bRunMinus				:= FALSE;
				arFlexoStation[i].bJog					:= FALSE;
				arFlexoStation[i].bStop					:= FALSE;
				arFlexoStation[i].bSetup				:= FALSE;
				arFlexoStation[i].bInkingOn				:= FALSE;
				arFlexoStation[i].bPrintingOn			:= FALSE;

				
	16#77:	//RUN SPD Minus

				arFlexoStation[i].bAniloxMtr 			:= FALSE;
				arFlexoStation[i].bAniloxKickOff 		:= FALSE;
				arFlexoStation[i].bPlateKickoff 		:= FALSE;
				arFlexoStation[i].bInfraRed 			:= FALSE;
				arFlexoStation[i].bRegAdvance			:= FALSE;
				arFlexoStation[i].bRegRetard			:= FALSE;
				arFlexoStation[i].bRunPlus				:= FALSE;
				arFlexoStation[i].bRunMinus				:= TRUE;
				arFlexoStation[i].bJog					:= FALSE;
				arFlexoStation[i].bStop					:= FALSE;
				arFlexoStation[i].bSetup				:= FALSE;
				arFlexoStation[i].bInkingOn				:= FALSE;
				arFlexoStation[i].bPrintingOn			:= FALSE;
				
	16#7B:	//RUN SPD Plus

				arFlexoStation[i].bAniloxMtr 			:= FALSE;
				arFlexoStation[i].bAniloxKickOff 		:= FALSE;
				arFlexoStation[i].bPlateKickoff 		:= FALSE;
				arFlexoStation[i].bInfraRed 			:= FALSE;
				arFlexoStation[i].bRegAdvance			:= FALSE;
				arFlexoStation[i].bRegRetard			:= FALSE;
				arFlexoStation[i].bRunPlus				:= TRUE;
				arFlexoStation[i].bRunMinus				:= FALSE;
				arFlexoStation[i].bJog					:= FALSE;
				arFlexoStation[i].bStop					:= FALSE;
				arFlexoStation[i].bSetup				:= FALSE;
				arFlexoStation[i].bInkingOn				:= FALSE;
				arFlexoStation[i].bPrintingOn			:= FALSE;
				
				
	16#DE:	//JOG

				arFlexoStation[i].bAniloxMtr 			:= FALSE;
				arFlexoStation[i].bAniloxKickOff 		:= FALSE;
				arFlexoStation[i].bPlateKickoff 		:= FALSE;
				arFlexoStation[i].bInfraRed 			:= FALSE;
				arFlexoStation[i].bRegAdvance			:= FALSE;
				arFlexoStation[i].bRegRetard			:= FALSE;
				arFlexoStation[i].bRunPlus				:= FALSE;
				arFlexoStation[i].bRunMinus				:= FALSE;
				arFlexoStation[i].bJog					:= TRUE;
				arFlexoStation[i].bStop					:= FALSE;
				arFlexoStation[i].bSetup				:= FALSE;
				arFlexoStation[i].bInkingOn				:= FALSE;
				arFlexoStation[i].bPrintingOn			:= FALSE;
				
	16#EE:	//STOP

				arFlexoStation[i].bAniloxMtr 			:= FALSE;
				arFlexoStation[i].bAniloxKickOff 		:= FALSE;
				arFlexoStation[i].bPlateKickoff 		:= FALSE;
				arFlexoStation[i].bInfraRed 			:= FALSE;
				arFlexoStation[i].bRegAdvance			:= FALSE;
				arFlexoStation[i].bRegRetard			:= FALSE;
				arFlexoStation[i].bRunPlus				:= FALSE;
				arFlexoStation[i].bRunMinus				:= FALSE;
				arFlexoStation[i].bJog					:= FALSE;
				arFlexoStation[i].bStop					:= TRUE;
				arFlexoStation[i].bSetup				:= FALSE;
				arFlexoStation[i].bInkingOn				:= FALSE;
				arFlexoStation[i].bPrintingOn			:= FALSE;
	
	ELSE
	
				arFlexoStation[i].bAniloxMtr 			:= FALSE;
				arFlexoStation[i].bAniloxKickOff 		:= FALSE;
				arFlexoStation[i].bPlateKickoff 		:= FALSE;
				arFlexoStation[i].bInfraRed 			:= FALSE;
				arFlexoStation[i].bRegAdvance			:= FALSE;
				arFlexoStation[i].bRegRetard			:= FALSE;
				arFlexoStation[i].bRunPlus				:= FALSE;
				arFlexoStation[i].bRunMinus				:= FALSE;
				arFlexoStation[i].bJog					:= FALSE;
				arFlexoStation[i].bStop					:= FALSE;
				arFlexoStation[i].bSetup				:= FALSE;
				arFlexoStation[i].bInkingOn				:= FALSE;
				arFlexoStation[i].bPrintingOn			:= FALSE;
	END_CASE;




END_FOR





bRun_gb	:=	arFlexoStation[1].bRunMinus OR arFlexoStation[1].bRunPlus OR arFlexoStation[2].bRunMinus OR arFlexoStation[2].bRunPlus	OR
			arFlexoStation[3].bRunMinus OR arFlexoStation[3].bRunPlus OR arFlexoStation[4].bRunMinus OR arFlexoStation[4].bRunPlus	OR
			arFlexoStation[5].bRunMinus OR arFlexoStation[5].bRunPlus OR arFlexoStation[6].bRunMinus OR arFlexoStation[6].bRunPlus	OR
			arFlexoStation[7].bRunMinus OR arFlexoStation[7].bRunPlus OR arFlexoStation[8].bRunMinus OR arFlexoStation[8].bRunPlus	OR
			arFlexoStation[9].bRunMinus OR arFlexoStation[9].bRunPlus OR arFlexoStation[10].bRunMinus OR arFlexoStation[10].bRunPlus OR
			arFlexoStation[11].bRunMinus OR arFlexoStation[11].bRunPlus OR arFlexoStation[12].bRunMinus OR arFlexoStation[12].bRunPlus OR
			arFlexoStation[13].bRunMinus OR arFlexoStation[13].bRunPlus OR arFlexoStation[14].bRunMinus OR arFlexoStation[14].bRunPlus OR		
			bRun_i;


//bRun_gb := bRunPlus_1 OR bRunMinus_1 OR bRunPlus_2 OR bRunMinus_2 OR bRunPlus_3 OR bRunMinus_3 OR bRunPlus_4 OR bRunMinus_4 OR bRunPlus_5 OR bRunMinus_5 

bResetSpeed_q := bRun_gb AND (NOT runOut);

//bJog_gb	:=  bJog_1 OR bJog_2 OR bJog_3 OR bJog_4 OR bJog_5 OR bJog_i;

//bJog_gb	:=  arFlexoStation[1].bJog;
bJog_gb	:=	arFlexoStation[1].bJog OR arFlexoStation[2].bJog OR arFlexoStation[3].bJog OR arFlexoStation[4].bJog OR 
				arFlexoStation[5].bJog OR arFlexoStation[6].bJog OR arFlexoStation[7].bJog OR arFlexoStation[8].bJog OR 
				arFlexoStation[9].bJog OR arFlexoStation[10].bJog OR arFlexoStation[11].bJog OR arFlexoStation[12].bJog OR
				arFlexoStation[13].bJog OR arFlexoStation[14].bJog  OR bJog_i;


bStop_gb	:=	arFlexoStation[1].bStop OR arFlexoStation[2].bStop OR arFlexoStation[3].bStop OR arFlexoStation[4].bStop OR 
				arFlexoStation[5].bStop OR arFlexoStation[6].bStop OR arFlexoStation[7].bStop OR arFlexoStation[8].bStop OR
				arFlexoStation[9].bStop OR arFlexoStation[10].bStop OR arFlexoStation[11].bStop OR arFlexoStation[12].bStop OR 
				arFlexoStation[13].bStop OR arFlexoStation[14].bStop  OR bStop_i;



bInkingOn_gb	:=	arFlexoStation[1].bInkingOn OR arFlexoStation[2].bInkingOn OR arFlexoStation[3].bInkingOn OR arFlexoStation[4].bInkingOn OR 
				arFlexoStation[5].bInkingOn OR arFlexoStation[6].bInkingOn OR arFlexoStation[7].bInkingOn OR arFlexoStation[8].bInkingOn OR 
				arFlexoStation[9].bInkingOn OR arFlexoStation[10].bInkingOn OR arFlexoStation[11].bInkingOn OR arFlexoStation[12].bInkingOn OR
				arFlexoStation[13].bInkingOn OR arFlexoStation[14].bInkingOn OR arFlexoStation[15].bInkingOn OR arFlexoStation[16].bInkingOn;
				
bPrintingOn_gb	:=	arFlexoStation[1].bPrintingOn OR arFlexoStation[2].bPrintingOn OR arFlexoStation[3].bPrintingOn OR arFlexoStation[4].bPrintingOn OR 
				arFlexoStation[5].bPrintingOn OR arFlexoStation[6].bPrintingOn OR arFlexoStation[7].bPrintingOn OR arFlexoStation[8].bPrintingOn OR 
				arFlexoStation[9].bPrintingOn OR arFlexoStation[10].bPrintingOn OR arFlexoStation[11].bPrintingOn OR arFlexoStation[12].bPrintingOn OR
				arFlexoStation[13].bPrintingOn OR arFlexoStation[14].bPrintingOn OR arFlexoStation[15].bPrintingOn OR arFlexoStation[16].bPrintingOn;


//bSetup_gb	:=	arFlexoStation[1].bSetup OR arFlexoStation[2].bSetup OR arFlexoStation[3].bSetup OR arFlexoStation[4].bSetup OR 
	//			arFlexoStation[5].bSetup OR arFlexoStation[6].bSetup OR arFlexoStation[7].bSetup OR arFlexoStation[8].bSetup OR 
	//			arFlexoStation[9].bSetup OR arFlexoStation[10].bSetup;

bComHealthy_gb	:=	(bComHeartBeat1_CAN_i OR bComHeartBeat1_Bypass_CAN_i) AND 
					(bComHeartBeat2_CAN_i OR bComHeartBeat2_Bypass_CAN_i) AND
					(bComHeartBeat3_CAN_i OR bComHeartBeat3_Bypass_CAN_i) AND
					(bComHeartBeat4_CAN_i OR bComHeartBeat4_Bypass_CAN_i) AND
					(bComHeartBeat5_CAN_i OR bComHeartBeat5_Bypass_CAN_i) AND
					(bComHeartBeat6_CAN_i OR bComHeartBeat6_Bypass_CAN_i) AND 
					(bComHeartBeat7_CAN_i OR bComHeartBeat7_Bypass_CAN_i) AND
					(bComHeartBeat8_CAN_i OR bComHeartBeat8_Bypass_CAN_i) ;
					
					(*(bComHeartBeat9_CAN_i OR bComHeartBeat9_Bypass_CAN_i) AND
					(bComHeartBeat10_CAN_i OR bComHeartBeat10_Bypass_CAN_i) AND
					(bComHeartBeat11_CAN_i OR bComHeartBeat11_Bypass_CAN_i) AND
					(bComHeartBeat12_CAN_i OR bComHeartBeat12_Bypass_CAN_i) AND
					(bComHeartBeat13_CAN_i OR bComHeartBeat13_Bypass_CAN_i);*)





IF bComHeartBeat1_CAN_i = TRUE THEN
	bComHeartBeat1_Bypass_CAN_i := FALSE;
END_IF

IF bComHeartBeat2_CAN_i = TRUE THEN
	bComHeartBeat2_Bypass_CAN_i := FALSE;
END_IF

IF bComHeartBeat3_CAN_i = TRUE THEN
	bComHeartBeat3_Bypass_CAN_i := FALSE;
END_IF

IF bComHeartBeat4_CAN_i = TRUE THEN
	bComHeartBeat4_Bypass_CAN_i := FALSE;
END_IF

IF bComHeartBeat5_CAN_i = TRUE THEN
	bComHeartBeat5_Bypass_CAN_i := FALSE;
END_IF

IF bComHeartBeat6_CAN_i = TRUE THEN
	bComHeartBeat6_Bypass_CAN_i := FALSE;
END_IF

IF bComHeartBeat7_CAN_i = TRUE THEN
	bComHeartBeat7_Bypass_CAN_i := FALSE;
END_IF

IF bComHeartBeat8_CAN_i = TRUE THEN
	bComHeartBeat8_Bypass_CAN_i := FALSE;
END_IF

IF bComHeartBeat9_CAN_i = TRUE THEN
	bComHeartBeat9_Bypass_CAN_i := FALSE;
END_IF

IF bComHeartBeat10_CAN_i = TRUE THEN
	bComHeartBeat10_Bypass_CAN_i := FALSE;
END_IF

IF bComHeartBeat11_CAN_i = TRUE THEN
	bComHeartBeat11_Bypass_CAN_i := FALSE;
END_IF

IF bComHeartBeat12_CAN_i = TRUE THEN
	bComHeartBeat12_Bypass_CAN_i := FALSE;
END_IF



bComHeartBeat1_CAN_i	:= STATION_BOARD1.bSlaveAvailable;
bComHeartBeat2_CAN_i	:= STATION_BOARD2.bSlaveAvailable;


//bComHeartBeatRelay1_CAN_i	:= RELAY_BOARD1.bSlaveAvailable;
//bComHeartBeatRelay2_CAN_i	:= RELAY_BOARD2.bSlaveAvailable;
//bComHeartBeatRelay3_CAN_i	:= RELAY_BOARD3.bSlaveAvailable;
//bComHeartBeatRelay4_CAN_i	:= RELAY_BOARD4.bSlaveAvailable;
//bComHeartBeatRelay5_CAN_i	:= RELAY_BOARD5.bSlaveAvailable;
//bComHeartBeatRelay6_CAN_i	:= RELAY_BOARD6.bSlaveAvailable;
//bComHeartBeatRelay7_CAN_i	:= RELAY_BOARD7.bSlaveAvailable;

END_PROGRAM

// MyController/Application/CONVERT
PROGRAM CONVERT
VAR
	
	dwDeviation_low_gb:DWORD;
	dwDeviation_high_gb:DWORD;
	dwDeviation_tot_gb:DWORD;
	rDeviation_gb:REAL;
	
	dwRegAdjustStep_low_gb:DWORD;
	dwRegAdjustStep_high_gb:DWORD;
	dwRegAdjustStep_tot_gb:DWORD;
	dwRegAdjustStep_gb:REAL;
	
	
	dwLoadcellTension_low_gb:DWORD;
	dwLoadcellTension_high_gb:DWORD;
	dwLoadcellTension_tot_gb:DWORD;
	rLoadcellTension_gb:REAL;
	
	dwRegiCtrlSetpoint_low_gb:DWORD;
	dwRegiCtrlSetpoint_high_gb:DWORD;
	dwRegiCtrlSetpoint_tot_gb:DWORD;
	rRegiCtrlSetpoint_gb:REAL;
END_VAR



GVL_CONVERT.bAnxMot_q1	:= ArFlexoStation[1].bAniloxMot_q;
GVL_CONVERT.bAnxMot_q2	:= ArFlexoStation[2].bAniloxMot_q;
GVL_CONVERT.bAnxMot_q3	:= ArFlexoStation[3].bAniloxMot_q;
GVL_CONVERT.bAnxMot_q4	:= ArFlexoStation[4].bAniloxMot_q;
GVL_CONVERT.bAnxMot_q5	:= ArFlexoStation[5].bAniloxMot_q;
GVL_CONVERT.bAnxMot_q6	:= ArFlexoStation[6].bAniloxMot_q;
GVL_CONVERT.bAnxMot_q7	:= ArFlexoStation[7].bAniloxMot_q;
GVL_CONVERT.bAnxMot_q8	:= ArFlexoStation[8].bAniloxMot_q;

GVL_CONVERT.bAnxKickoff_q1	:= ArFlexoStation[1].bAniloxKickoff_q;
GVL_CONVERT.bAnxKickoff_q2	:= ArFlexoStation[2].bAniloxKickoff_q;
GVL_CONVERT.bAnxKickoff_q3	:= ArFlexoStation[3].bAniloxKickoff_q;
GVL_CONVERT.bAnxKickoff_q4	:= ArFlexoStation[4].bAniloxKickoff_q;
GVL_CONVERT.bAnxKickoff_q5	:= ArFlexoStation[5].bAniloxKickoff_q;
GVL_CONVERT.bAnxKickoff_q6	:= ArFlexoStation[6].bAniloxKickoff_q;
GVL_CONVERT.bAnxKickoff_q7	:= ArFlexoStation[7].bAniloxKickoff_q;
GVL_CONVERT.bAnxKickoff_q8	:= ArFlexoStation[8].bAniloxKickoff_q;


GVL_CONVERT.bPlateKickoff_q1	:= ArFlexoStation[1].bPlateKickoff_q;
GVL_CONVERT.bPlateKickoff_q2	:= ArFlexoStation[2].bPlateKickoff_q;
GVL_CONVERT.bPlateKickoff_q3	:= ArFlexoStation[3].bPlateKickoff_q;
GVL_CONVERT.bPlateKickoff_q4	:= ArFlexoStation[4].bPlateKickoff_q;
GVL_CONVERT.bPlateKickoff_q5	:= ArFlexoStation[5].bPlateKickoff_q;
GVL_CONVERT.bPlateKickoff_q6	:= ArFlexoStation[6].bPlateKickoff_q;
GVL_CONVERT.bPlateKickoff_q7	:= ArFlexoStation[7].bPlateKickoff_q;
GVL_CONVERT.bPlateKickoff_q8	:= ArFlexoStation[8].bPlateKickoff_q;


GVL_CONVERT.bRegAdv_q1	:= ArFlexoStation[1].bRegAdvance;
GVL_CONVERT.bRegAdv_q2	:= ArFlexoStation[2].bRegAdvance;
GVL_CONVERT.bRegAdv_q3	:= ArFlexoStation[3].bRegAdvance;
GVL_CONVERT.bRegAdv_q4	:= ArFlexoStation[4].bRegAdvance;
GVL_CONVERT.bRegAdv_q5	:= ArFlexoStation[5].bRegAdvance;
GVL_CONVERT.bRegAdv_q6	:= ArFlexoStation[6].bRegAdvance;
GVL_CONVERT.bRegAdv_q7	:= ArFlexoStation[7].bRegAdvance;
GVL_CONVERT.bRegAdv_q8	:= ArFlexoStation[8].bRegAdvance;


GVL_CONVERT.bRegRet_q1	:= ArFlexoStation[1].bRegRetard;
GVL_CONVERT.bRegRet_q2	:= ArFlexoStation[2].bRegRetard;
GVL_CONVERT.bRegRet_q3	:= ArFlexoStation[3].bRegRetard;
GVL_CONVERT.bRegRet_q4	:= ArFlexoStation[4].bRegRetard;
GVL_CONVERT.bRegRet_q5	:= ArFlexoStation[5].bRegRetard;
GVL_CONVERT.bRegRet_q6	:= ArFlexoStation[6].bRegRetard;
GVL_CONVERT.bRegRet_q7	:= ArFlexoStation[7].bRegRetard;
GVL_CONVERT.bRegRet_q8	:= ArFlexoStation[8].bRegRetard;


//uiDeviation_low_gb + uiDeviation_high_gb
dwDeviation_high_gb	:=	SHL(wDeviation_high_gb,16);
dwDeviation_low_gb	:=	wDeviation_low_gb;
dwDeviation_tot_gb	:=	dwDeviation_low_gb OR dwDeviation_high_gb;
rDeviation_gb:= (DWORD_TO_REAL(dwDeviation_tot_gb)/100000)-360.0;
rDeviation_HMI_q	:=	rDeviation_gb;

dwLoadcellTension_high_gb	:=	SHL(wLoadcellTension_high_gb,16);
dwLoadcellTension_low_gb	:=	wLoadcellTension_low_gb;
dwLoadcellTension_tot_gb	:=	dwLoadcellTension_low_gb OR dwLoadcellTension_high_gb;
rLoadcellTension_gb:= (DWORD_TO_REAL((dwLoadcellTension_tot_gb*60)/1000));
bInfeed_Tension_HMI	:=	rLoadcellTension_gb;

//rRegAdjustStep_HMI_i

IF rRegAdjustStep_HMI_i = 0.0 THEN
	rRegAdjustStep_HMI_i := 100.0;
END_IF
dwRegAdjustStep_tot_gb :=	REAL_TO_DWORD(rRegAdjustStep_HMI_i*1000.0);
dwRegAdjustStep_high_gb	:=	SHR(dwRegAdjustStep_tot_gb,16);
dwRegAdjustStep_low_gb := dwRegAdjustStep_tot_gb AND 65535;
wRegAdjustStep_high_gb := DWORD_TO_WORD(dwRegAdjustStep_high_gb);
wRegAdjustStep_low_gb := DWORD_TO_WORD(dwRegAdjustStep_low_gb);

wInfeedManualGearing_HMI_i := WORD_to_UINT(wInfeedManualGearing_ETH_i);

//wRegiCtrlSetpoint_low_gb
dwRegiCtrlSetpoint_high_gb	:=	SHL(wRegiCtrlSetpoint_high_gb,16);
dwRegiCtrlSetpoint_low_gb	:=	wRegiCtrlSetpoint_low_gb;
dwRegiCtrlSetpoint_tot_gb	:=	dwRegiCtrlSetpoint_low_gb OR dwRegiCtrlSetpoint_high_gb;
rRegiCtrlSetpoint_gb:= (DWORD_TO_REAL(dwRegiCtrlSetpoint_tot_gb)/100000)-360.0;
//rDeviation_HMI_q	:=	rDeviation_gb;
rRegiCtrlSetpoint_HMI_q	:=	rRegiCtrlSetpoint_gb;

END_PROGRAM

// MyController/Application/DRYER_1FD_3FX_STATIONS
PROGRAM DRYER_1FD_3FX_STATIONS
VAR
	uiBogus:UINT;
	fbIR1_Delay: TON;
	fbIR1_Low_Delay: TON;
	fbIR2_Low_Delay: TON;
	
	fbIR1_High_Delay: TON;
	fbIR2_High_Delay: TON;
	
	fbIR3_Low_Delay: TON;
	fbIR4_Low_Delay: TON;
	
	fbIR5_Low_Delay: TON;
	fbIR6_Low_Delay: TON;
	fbIR7_Low_Delay: TON;
	fbIR8_Low_Delay: TON;
	fbIR9_Low_Delay: TON;
	fbIR10_Low_Delay: TON;

	fbIR3_High_Delay: TON;
	fbIR4_High_Delay: TON;
	
	tElapsedTimeLow1:TIME;
	tElapsedTimeHigh1:TIME;
	
	tElapsedTimeLow2:TIME;
	tElapsedTimeHigh2:TIME;
	
	tElapsedTimeLow3:TIME;
	tElapsedTimeHigh3:TIME;
	
    tElapsedTimeLow4:TIME;
	tElapsedTimeHigh4:TIME;	
	
	tElapsedTimeLow5:TIME;
	tElapsedTimeLow6:TIME;
	tElapsedTimeLow7:TIME;
	tElapsedTimeLow8:TIME;
	tElapsedTimeLow9:TIME;
	tElapsedTimeLow10:TIME;
	
	tElapsedTimeCheck1:TIME;
	tElapsedTimeCheck2:TIME;
	tElapsedTimeCheck3:TIME;
	tElapsedTimeCheck4:TIME;
	tElapsedTimeCheck5:TIME;
	

	
	fbHeatEnable1: TON;
	fbHeatEnable2: TON;
	fbHeatEnable3: TON;
	fbHeatEnable4: TON;
    fbHeatEnable5: TON;
	
	
	bAbortGroup1:BOOL := FALSE;
	bAbortGroup2:BOOL := FALSE;
	bAbortGroup3:BOOL := FALSE;
	bAbortGroup4:BOOL := FALSE;
	bAbortGroup5:BOOL := FALSE;
	bAbortGroup6:BOOL := FALSE;
	
	fb_ABORTGROUP1_KEEP: SR;
	fb_ABORTGROUP2_KEEP: SR;
	fb_ABORTGROUP3_KEEP: SR;
	fb_ABORTGROUP4_KEEP: SR;
	fb_ABORTGROUP5_KEEP: SR;
	fb_ABORTGROUP6_KEEP: SR;
	
	bSomethingOn:BOOL;
	fbHeatGroup1_Delay: TON;

	fbHeatEnable6: TON;
	SR_FD6: SR;
	timerFD6: TON;
	tElapsedTimeCheck6: TIME;
	
